VAR_TEMP
  iRetVal : INT ;	//return value as integer
  wRetVal : WORD ;	//return value as word
  Run : BOOL ;	//Unit in "RUN" mode
  EStopOK : BOOL ;	//Emergency Stop OK
  CIP : BOOL ;	//CIP Program Selected
  ComCIP : BOOL ;	//Communication with CIP Active
  xTmp : BOOL ;	//Temporary BOOL (free for general use)
  iTmp : INT ;	//Temporary INT (free for general use)
  rTmp : REAL ;	//Temporary REAL (free for general use)
  dTmp : DINT ;	//Temporary DINT (free for general use)
  UnitNo : INT ;	//Unit Number
  EquipmentID : INT ;	//Equipment ID
  Prid : DINT ;	//Process ID
  SFM36 : STRUCT 	// CIP Pump Mode
   I00 : BOOL ;	// Off
   I01 : BOOL ;	// Flow
   I02 : BOOL ;	// Pressure
   I03 : BOOL ;	// Fix Speed
   I04 : BOOL ;
   I05 : BOOL ;
   I06 : BOOL ;
   I07 : BOOL ;
   I08 : BOOL ;
   I09 : BOOL ;
   I10 : BOOL ;
   I11 : BOOL ;
   I12 : BOOL ;
   I13 : BOOL ;
   I14 : BOOL ;
   I15 : BOOL ;
   I16 : BOOL ;
   I17 : BOOL ;
   I18 : BOOL ;
   I19 : BOOL ;
   I20 : BOOL ;
   I21 : BOOL ;
   I22 : BOOL ;
   I23 : BOOL ;
   I24 : BOOL ;
   I25 : BOOL ;
   I26 : BOOL ;
   I27 : BOOL ;
   I28 : BOOL ;
   I29 : BOOL ;
   I30 : BOOL ;
   I31 : BOOL ;
  END_STRUCT ;
END_VAR
BEGIN
NETWORK
TITLE =general

      SET   ;

// unit & equipment number ---------------------------------------------------
      L     DB4210.DBW    0;
      T     #UnitNo;

      L     DB4215.DBW   14;
      L     1000;
      *I    ;
      L     #UnitNo;
      +I    ;
      T     #EquipmentID;

// CIP ----------------------------------------------------------------------
      L     DB4215.DBW   18;
      L     0;
      <I    ;
      =     #CIP;

// Communicating Units-------------------------------------------------------
      L     DB4215.DBD   10;
      L     DB4215.DBD  106;
      ==D   ;
      =     #ComCIP;

// emergency OK -------------------------------------------------------------
      A     DB4215.DBX   75.0; //General Emergency Stop OK
      CLR   ;
      =     #EStopOK;

NETWORK
TITLE =read other unit's data

      SET   ;

// ... General Unit ----------/

      CALL FC   563 (
           ActReq                   := M    101.0,
           PLCNo                    := 3,
           SourceUnitNo             := 99,
           IsTUnit                  := FALSE,
           DstComDRec               := DB4215.GEN,
           RET_VAL                  := #wRetVal);


NETWORK
TITLE =remote start

      SET   ;
// !!! insert correct condition of unit start !!!
      A     DB4211.DBX   15.0;
      A     DB4211.DBX   17.4;
      CLR   ;
      JCN   Strt;
      L     DB4215.DBD   10;
//L        L#-1;                            // Prid negative to start on its own
      T     #Prid;

      CALL FC    48 (
           UnitNo                   := #UnitNo,
           PrId                     := #Prid,
           Run                      := DB4211.DBX   17.4,
           PrIdTransfer             := TRUE,
           Start                    := TRUE,
           RetVal                   := #wRetVal);
Strt: NOP   0;
NETWORK
TITLE =external releases

      SET   ;

NETWORK
TITLE =write own unit data

      SET   ;

//-- CIP Communication ---------------------------------------
      AN    DB4211.DBX   15.0;
//      AN "U121SeqD".Seq.PO.B30 // CIP Active (Slave)
      A     #ComCIP;
      JCN   NCIP;
//Conductivity CIP Return
      L     DB4215.DBD  150;
      T     DB4211.DBD  626;

//Temperature CIP Return
      L     DB4215.DBD  146;
      T     DB4211.DBD  594;

//CIP Prerun Pump SP

      CALL FC    45 (
           SFM                      := DB4211.DBD  686,
           Indexes                  := #SFM36);


      L     0.000000e+000;
      A     #SFM36.I01;
      =     DB4215.DBX  171.7;
      JCN   pfc;
      L     DB4211.DBD  654;
pfc:  NOP   0;
      A     #SFM36.I02;
      =     DB4215.DBX  172.0;
      JCN   ppc;
      L     DB4211.DBD  670;
ppc:  NOP   0;
      A     #SFM36.I03;
      =     DB4215.DBX  171.6;
      JCN   pxc;
      L     DB4211.DBD  574;
pxc:  NOP   0;
      T     DB4215.DBD  182;

//CIP Return
      L     DB4211.DBD  558;
      T     DB4215.DBD  186;
      L     DB4215.DBD  138;
      T     DB4211.DBD  562;

//CIP Prerun
      L     DB4211.DBD  542;
      T     DB4215.DBD  190;
      L     DB4215.DBD  142;
      T     DB4211.DBD  546;

// Write Own Data to CIP
      L     DB4215.DBD   10;
      T     DB4215.DBD  154;

      L     DB4215.DBW   14;
      T     DB4215.DBW  158;

      L     DB4215.DBW   16;
      T     DB4215.DBW  160;

      L     DB4215.DBW   18;
      T     DB4215.DBW  162;

      L     DB4215.DBW   20;
      T     DB4215.DBW  164;

      L     DB4215.DBW   22;
      T     DB4215.DBW  166;

      A     DB4215.DBX   24.0;
      =     DB4215.DBX  168.0;

      A     DB4215.DBX   24.1;
      =     DB4215.DBX  168.1;

      A     DB4215.DBX   24.2;
      =     DB4215.DBX  168.2;

      A     DB4215.DBX   24.3;
      =     DB4215.DBX  168.3;

      A     DB4215.DBX   24.4;
      =     DB4215.DBX  168.4;

      A     DB4215.DBX   24.5;
      =     DB4215.DBX  168.5;

      A     DB4215.DBX   24.6;
      =     DB4215.DBX  168.6;

      A     DB4215.DBX   24.7;
      =     DB4215.DBX  168.7;

// Copy Data to CIP
      CALL SFC   20 (
           SRCBLK                   := DB4215.ToCIP,
           RET_VAL                  := #iRetVal,
           DSTBLK                   := DB4215.ToCIP);

NCIP: NOP   0;

//Empty Signal
//A     "U121SpID".SpI.Sig //!!!! Insert correct Empty Signal !!!
      CLR   ;
      =     DB4215.DBX   26.5;

//Full Signal
//A     "U121SpID".SpI.Sig //!!!! Insert correct Full Signal !!!
      CLR   ;
      =     DB4215.DBX   26.2;

//CIP Program Selected
      A     #CIP;
      =     DB4215.DBX   27.1;

// Emergency Stop
      A     #EStopOK; //If needed add or replace with own SpI
      =     DB4215.DBX   27.0; //Emergency Stop OK


NETWORK
TITLE = read from other unit data



END_FUNCTION_BLOCK

FUNCTION_BLOCK FB 4225
TITLE =U122: Planung Transfer VE2
FAMILY : BOTEC_F1
NAME : U122Comm
VERSION : 0.1


VAR_TEMP
  iRetVal : INT ;	//return value as integer
  wRetVal : WORD ;	//return value as word
  Run : BOOL ;	//Unit in "RUN" mode
  EStopOK : BOOL ;	//Emergency Stop OK
  CIP : BOOL ;	//CIP Program Selected
  ComCIP : BOOL ;	//Communication with CIP Active
  xTmp : BOOL ;	//Temporary BOOL (free for general use)
  iTmp : INT ;	//Temporary INT (free for general use)
  rTmp : REAL ;	//Temporary REAL (free for general use)
  dTmp : DINT ;	//Temporary DINT (free for general use)
  UnitNo : INT ;	//Unit Number
  EquipmentID : INT ;	//Equipment ID
  Prid : DINT ;	//Process ID
  SFM36 : STRUCT 	// CIP Pump Mode
   I00 : BOOL ;	// Off
   I01 : BOOL ;	// Flow
   I02 : BOOL ;	// Pressure
   I03 : BOOL ;	// Fix Speed
   I04 : BOOL ;
   I05 : BOOL ;
   I06 : BOOL ;
   I07 : BOOL ;
   I08 : BOOL ;
   I09 : BOOL ;
   I10 : BOOL ;
   I11 : BOOL ;
   I12 : BOOL ;
   I13 : BOOL ;
   I14 : BOOL ;
   I15 : BOOL ;
   I16 : BOOL ;
   I17 : BOOL ;
   I18 : BOOL ;
   I19 : BOOL ;
   I20 : BOOL ;
   I21 : BOOL ;
   I22 : BOOL ;
   I23 : BOOL ;
   I24 : BOOL ;
   I25 : BOOL ;
   I26 : BOOL ;
   I27 : BOOL ;
   I28 : BOOL ;
   I29 : BOOL ;
   I30 : BOOL ;
   I31 : BOOL ;
  END_STRUCT ;
END_VAR
BEGIN
NETWORK
TITLE =general

      SET   ;

// unit & equipment number ---------------------------------------------------
      L     DB4220.DBW    0;
      T     #UnitNo;

      L     DB4225.DBW   14;
      L     1000;
      *I    ;
      L     #UnitNo;
      +I    ;
      T     #EquipmentID;

// CIP ----------------------------------------------------------------------
      L     DB4225.DBW   18;
      L     0;
      <I    ;
      =     #CIP;

// Communicating Units-------------------------------------------------------
      L     DB4225.DBD   10;
      L     DB4225.DBD  106;
      ==D   ;
      =     #ComCIP;

// emergency OK -------------------------------------------------------------
      A     DB4225.DBX   75.0; //General Emergency Stop OK
      CLR   ;
      =     #EStopOK;

NETWORK
TITLE =read other unit's data

      SET   ;

// ... General Unit ----------/

      CALL FC   563 (
           ActReq                   := M    101.0,
           PLCNo                    := 3,
           SourceUnitNo             := 99,
           IsTUnit                  := FALSE,
           DstComDRec               := DB4225.GEN,
           RET_VAL                  := #wRetVal);

NETWORK
TITLE =remote start

      SET   ;
// !!! insert correct condition of unit start !!!
      A     DB4221.DBX   15.0;
      A     DB4221.DBX   17.4;
      CLR   ;
      JCN   Strt;
      L     DB4225.DBD   10;
//L        L#-1;                            // Prid negative to start on its own
      T     #Prid;

      CALL FC    48 (
           UnitNo                   := #UnitNo,
           PrId                     := #Prid,
           Run                      := DB4221.DBX   17.4,
           PrIdTransfer             := TRUE,
           Start                    := TRUE,
           RetVal                   := #wRetVal);
Strt: NOP   0;
NETWORK
TITLE =external releases

      SET   ;

NETWORK
TITLE =write own unit data

      SET   ;

//-- CIP Communication ---------------------------------------
      AN    DB4221.DBX   15.0;
//      AN "U122SeqD".Seq.PO.B30 // CIP Active (Slave)
      A     #ComCIP;
      JCN   NCIP;
//Conductivity CIP Return
      L     DB4225.DBD  150;
      T     DB4221.DBD  626;

//Temperature CIP Return
      L     DB4225.DBD  146;
      T     DB4221.DBD  594;

//CIP Prerun Pump SP

      CALL FC    45 (
           SFM                      := DB4221.DBD  686,
           Indexes                  := #SFM36);


      L     0.000000e+000;
      A     #SFM36.I01;
      =     DB4225.DBX  171.7;
      JCN   pfc;
      L     DB4221.DBD  654;
pfc:  NOP   0;
      A     #SFM36.I02;
      =     DB4225.DBX  172.0;
      JCN   ppc;
      L     DB4221.DBD  670;
ppc:  NOP   0;
      A     #SFM36.I03;
      =     DB4225.DBX  171.6;
      JCN   pxc;
      L     DB4221.DBD  574;
pxc:  NOP   0;
      T     DB4225.DBD  182;

//CIP Return
      L     DB4221.DBD  558;
      T     DB4225.DBD  186;
      L     DB4225.DBD  138;
      T     DB4221.DBD  562;

//CIP Prerun
      L     DB4221.DBD  542;
      T     DB4225.DBD  190;
      L     DB4225.DBD  142;
      T     DB4221.DBD  546;

// Write Own Data to CIP
      L     DB4225.DBD   10;
      T     DB4225.DBD  154;

      L     DB4225.DBW   14;
      T     DB4225.DBW  158;

      L     DB4225.DBW   16;
      T     DB4225.DBW  160;

      L     DB4225.DBW   18;
      T     DB4225.DBW  162;

      L     DB4225.DBW   20;
      T     DB4225.DBW  164;

      L     DB4225.DBW   22;
      T     DB4225.DBW  166;

      A     DB4225.DBX   24.0;
      =     DB4225.DBX  168.0;

      A     DB4225.DBX   24.1;
      =     DB4225.DBX  168.1;

      A     DB4225.DBX   24.2;
      =     DB4225.DBX  168.2;

      A     DB4225.DBX   24.3;
      =     DB4225.DBX  168.3;

      A     DB4225.DBX   24.4;
      =     DB4225.DBX  168.4;

      A     DB4225.DBX   24.5;
      =     DB4225.DBX  168.5;

      A     DB4225.DBX   24.6;
      =     DB4225.DBX  168.6;

      A     DB4225.DBX   24.7;
      =     DB4225.DBX  168.7;

// Copy Data to CIP
      CALL SFC   20 (
           SRCBLK                   := DB4225.ToCIP,
           RET_VAL                  := #iRetVal,
           DSTBLK                   := DB4225.ToCIP);

NCIP: NOP   0;

//Empty Signal
//A     "U122SpID".SpI.Sig //!!!! Insert correct Empty Signal !!!
      CLR   ;
      =     DB4225.DBX   26.5;

//Full Signal
//A     "U122SpID".SpI.Sig //!!!! Insert correct Full Signal !!!
      CLR   ;
      =     DB4225.DBX   26.2;

//CIP Program Selected
      A     #CIP;
      =     DB4225.DBX   27.1;

// Emergency Stop
      A     #EStopOK; //If needed add or replace with own SpI
      =     DB4225.DBX   27.0; //Emergency Stop OK


NETWORK
TITLE = read from other unit data



END_FUNCTION_BLOCK

FUNCTION_BLOCK FB 4255
TITLE =U125: Planung Transfer A
FAMILY : BOTEC_F1
NAME : U125Comm
VERSION : 0.1


VAR_TEMP
  iRetVal : INT ;	//return value as integer
  wRetVal : WORD ;	//return value as word
  Run : BOOL ;	//Unit in "RUN" mode
  EStopOK : BOOL ;	//Emergency Stop OK
  CIP : BOOL ;	//CIP Program Selected
  ComCIP : BOOL ;	//Communication with CIP Active
  xTmp : BOOL ;	//Temporary BOOL (free for general use)
  iTmp : INT ;	//Temporary INT (free for general use)
  rTmp : REAL ;	//Temporary REAL (free for general use)
  dTmp : DINT ;	//Temporary DINT (free for general use)
  UnitNo : INT ;	//Unit Number
  EquipmentID : INT ;	//Equipment ID
  Prid : DINT ;	//Process ID
  SFM36 : STRUCT 	// CIP Pump Mode
   I00 : BOOL ;	// Off
   I01 : BOOL ;	// Flow
   I02 : BOOL ;	// Pressure
   I03 : BOOL ;	// Fix Speed
   I04 : BOOL ;
   I05 : BOOL ;
   I06 : BOOL ;
   I07 : BOOL ;
   I08 : BOOL ;
   I09 : BOOL ;
   I10 : BOOL ;
   I11 : BOOL ;
   I12 : BOOL ;
   I13 : BOOL ;
   I14 : BOOL ;
   I15 : BOOL ;
   I16 : BOOL ;
   I17 : BOOL ;
   I18 : BOOL ;
   I19 : BOOL ;
   I20 : BOOL ;
   I21 : BOOL ;
   I22 : BOOL ;
   I23 : BOOL ;
   I24 : BOOL ;
   I25 : BOOL ;
   I26 : BOOL ;
   I27 : BOOL ;
   I28 : BOOL ;
   I29 : BOOL ;
   I30 : BOOL ;
   I31 : BOOL ;
  END_STRUCT ;
END_VAR
BEGIN
NETWORK
TITLE =general

      SET   ;

// unit & equipment number ---------------------------------------------------
      L     DB4250.DBW    0;
      T     #UnitNo;

      L     DB4255.DBW   14;
      L     1000;
      *I    ;
      L     #UnitNo;
      +I    ;
      T     #EquipmentID;

// CIP ----------------------------------------------------------------------
      L     DB4255.DBW   18;
      L     0;
      <I    ;
      =     #CIP;

// Communicating Units-------------------------------------------------------
      L     DB4255.DBD   10;
      L     DB4255.DBD  106;
      ==D   ;
      =     #ComCIP;

// emergency OK -------------------------------------------------------------
      A     DB4255.DBX   75.0; //General Emergency Stop OK
      CLR   ;
      =     #EStopOK;

NETWORK
TITLE =read other unit's data

      SET   ;

// ... General Unit ----------/

      CALL FC   563 (
           ActReq                   := M    101.0,
           PLCNo                    := 3,
           SourceUnitNo             := 99,
           IsTUnit                  := FALSE,
           DstComDRec               := DB4255.GEN,
           RET_VAL                  := #wRetVal);

NETWORK
TITLE =remote start

      SET   ;
// !!! insert correct condition of unit start !!!
      A     DB4251.DBX   15.0;
      A     DB4251.DBX   17.4;
      CLR   ;
      JCN   Strt;
      L     DB4255.DBD   10;
//L        L#-1;                            // Prid negative to start on its own
      T     #Prid;

      CALL FC    48 (
           UnitNo                   := #UnitNo,
           PrId                     := #Prid,
           Run                      := DB4251.DBX   17.4,
           PrIdTransfer             := TRUE,
           Start                    := TRUE,
           RetVal                   := #wRetVal);
Strt: NOP   0;
NETWORK
TITLE =external releases

      SET   ;

NETWORK
TITLE =write own unit data

      SET   ;

//-- CIP Communication ---------------------------------------
      AN    DB4251.DBX   15.0;
//      AN "U125SeqD".Seq.PO.B30 // CIP Active (Slave)
      A     #ComCIP;
      JCN   NCIP;
//Conductivity CIP Return
      L     DB4255.DBD  150;
      T     DB4251.DBD  626;

//Temperature CIP Return
      L     DB4255.DBD  146;
      T     DB4251.DBD  594;

//CIP Prerun Pump SP

      CALL FC    45 (
           SFM                      := DB4251.DBD  686,
           Indexes                  := #SFM36);


      L     0.000000e+000;
      A     #SFM36.I01;
      =     DB4255.DBX  171.7;
      JCN   pfc;
      L     DB4251.DBD  654;
pfc:  NOP   0;
      A     #SFM36.I02;
      =     DB4255.DBX  172.0;
      JCN   ppc;
      L     DB4251.DBD  670;
ppc:  NOP   0;
      A     #SFM36.I03;
      =     DB4255.DBX  171.6;
      JCN   pxc;
      L     DB4251.DBD  574;
pxc:  NOP   0;
      T     DB4255.DBD  182;

//CIP Return
      L     DB4251.DBD  558;
      T     DB4255.DBD  186;
      L     DB4255.DBD  138;
      T     DB4251.DBD  562;

//CIP Prerun
      L     DB4251.DBD  542;
      T     DB4255.DBD  190;
      L     DB4255.DBD  142;
      T     DB4251.DBD  546;

// Write Own Data to CIP
      L     DB4255.DBD   10;
      T     DB4255.DBD  154;

      L     DB4255.DBW   14;
      T     DB4255.DBW  158;

      L     DB4255.DBW   16;
      T     DB4255.DBW  160;

      L     DB4255.DBW   18;
      T     DB4255.DBW  162;

      L     DB4255.DBW   20;
      T     DB4255.DBW  164;

      L     DB4255.DBW   22;
      T     DB4255.DBW  166;

      A     DB4255.DBX   24.0;
      =     DB4255.DBX  168.0;

      A     DB4255.DBX   24.1;
      =     DB4255.DBX  168.1;

      A     DB4255.DBX   24.2;
      =     DB4255.DBX  168.2;

      A     DB4255.DBX   24.3;
      =     DB4255.DBX  168.3;

      A     DB4255.DBX   24.4;
      =     DB4255.DBX  168.4;

      A     DB4255.DBX   24.5;
      =     DB4255.DBX  168.5;

      A     DB4255.DBX   24.6;
      =     DB4255.DBX  168.6;

      A     DB4255.DBX   24.7;
      =     DB4255.DBX  168.7;

// Copy Data to CIP
      CALL SFC   20 (
           SRCBLK                   := DB4255.ToCIP,
           RET_VAL                  := #iRetVal,
           DSTBLK                   := DB4255.ToCIP);

NCIP: NOP   0;

//Empty Signal
//A     "U125SpID".SpI.Sig //!!!! Insert correct Empty Signal !!!
      CLR   ;
      =     DB4255.DBX   26.5;

//Full Signal
//A     "U125SpID".SpI.Sig //!!!! Insert correct Full Signal !!!
      CLR   ;
      =     DB4255.DBX   26.2;

//CIP Program Selected
      A     #CIP;
      =     DB4255.DBX   27.1;

// Emergency Stop
      A     #EStopOK; //If needed add or replace with own SpI
      =     DB4255.DBX   27.0; //Emergency Stop OK


NETWORK
TITLE = read from other unit data



END_FUNCTION_BLOCK

FUNCTION_BLOCK FB 4265
TITLE =U126: Planung Transfer B
FAMILY : BOTEC_F1
NAME : U126Comm
VERSION : 0.1


VAR_TEMP
  iRetVal : INT ;	//return value as integer
  wRetVal : WORD ;	//return value as word
  Run : BOOL ;	//Unit in "RUN" mode
  EStopOK : BOOL ;	//Emergency Stop OK
  CIP : BOOL ;	//CIP Program Selected
  ComCIP : BOOL ;	//Communication with CIP Active
  xTmp : BOOL ;	//Temporary BOOL (free for general use)
  iTmp : INT ;	//Temporary INT (free for general use)
  rTmp : REAL ;	//Temporary REAL (free for general use)
  dTmp : DINT ;	//Temporary DINT (free for general use)
  UnitNo : INT ;	//Unit Number
  EquipmentID : INT ;	//Equipment ID
  Prid : DINT ;	//Process ID
  SFM36 : STRUCT 	// CIP Pump Mode
   I00 : BOOL ;	// Off
   I01 : BOOL ;	// Flow
   I02 : BOOL ;	// Pressure
   I03 : BOOL ;	// Fix Speed
   I04 : BOOL ;
   I05 : BOOL ;
   I06 : BOOL ;
   I07 : BOOL ;
   I08 : BOOL ;
   I09 : BOOL ;
   I10 : BOOL ;
   I11 : BOOL ;
   I12 : BOOL ;
   I13 : BOOL ;
   I14 : BOOL ;
   I15 : BOOL ;
   I16 : BOOL ;
   I17 : BOOL ;
   I18 : BOOL ;
   I19 : BOOL ;
   I20 : BOOL ;
   I21 : BOOL ;
   I22 : BOOL ;
   I23 : BOOL ;
   I24 : BOOL ;
   I25 : BOOL ;
   I26 : BOOL ;
   I27 : BOOL ;
   I28 : BOOL ;
   I29 : BOOL ;
   I30 : BOOL ;
   I31 : BOOL ;
  END_STRUCT ;
END_VAR
BEGIN
NETWORK
TITLE =general

      SET   ;

// unit & equipment number ---------------------------------------------------
      L     DB4260.DBW    0;
      T     #UnitNo;

      L     DB4265.DBW   14;
      L     1000;
      *I    ;
      L     #UnitNo;
      +I    ;
      T     #EquipmentID;

// CIP ----------------------------------------------------------------------
      L     DB4265.DBW   18;
      L     0;
      <I    ;
      =     #CIP;

// Communicating Units-------------------------------------------------------
      L     DB4265.DBD   10;
      L     DB4265.DBD  106;
      ==D   ;
      =     #ComCIP;

// emergency OK -------------------------------------------------------------
      A     DB4265.DBX   75.0; //General Emergency Stop OK
      CLR   ;
      =     #EStopOK;

NETWORK
TITLE =read other unit's data

      SET   ;

// ... General Unit ----------/

      CALL FC   563 (
           ActReq                   := M    101.0,
           PLCNo                    := 3,
           SourceUnitNo             := 99,
           IsTUnit                  := FALSE,
           DstComDRec               := DB4265.GEN,
           RET_VAL                  := #wRetVal);


NETWORK
TITLE =remote start

      SET   ;
// !!! insert correct condition of unit start !!!
      A     DB4261.DBX   15.0;
      A     DB4261.DBX   17.4;
      CLR   ;
      JCN   Strt;
      L     DB4265.DBD   10;
//L        L#-1;                            // Prid negative to start on its own
      T     #Prid;

      CALL FC    48 (
           UnitNo                   := #UnitNo,
           PrId                     := #Prid,
           Run                      := DB4261.DBX   17.4,
           PrIdTransfer             := TRUE,
           Start                    := TRUE,
           RetVal                   := #wRetVal);
Strt: NOP   0;
NETWORK
TITLE =external releases

      SET   ;

NETWORK
TITLE =write own unit data

      SET   ;

//-- CIP Communication ---------------------------------------
      AN    DB4261.DBX   15.0;
//      AN "U126SeqD".Seq.PO.B30 // CIP Active (Slave)
      A     #ComCIP;
      JCN   NCIP;
//Conductivity CIP Return
      L     DB4265.DBD  150;
      T     DB4261.DBD  626;

//Temperature CIP Return
      L     DB4265.DBD  146;
      T     DB4261.DBD  594;

//CIP Prerun Pump SP

      CALL FC    45 (
           SFM                      := DB4261.DBD  686,
           Indexes                  := #SFM36);


      L     0.000000e+000;
      A     #SFM36.I01;
      =     DB4265.DBX  171.7;
      JCN   pfc;
      L     DB4261.DBD  654;
pfc:  NOP   0;
      A     #SFM36.I02;
      =     DB4265.DBX  172.0;
      JCN   ppc;
      L     DB4261.DBD  670;
ppc:  NOP   0;
      A     #SFM36.I03;
      =     DB4265.DBX  171.6;
      JCN   pxc;
      L     DB4261.DBD  574;
pxc:  NOP   0;
      T     DB4265.DBD  182;

//CIP Return
      L     DB4261.DBD  558;
      T     DB4265.DBD  186;
      L     DB4265.DBD  138;
      T     DB4261.DBD  562;

//CIP Prerun
      L     DB4261.DBD  542;
      T     DB4265.DBD  190;
      L     DB4265.DBD  142;
      T     DB4261.DBD  546;

// Write Own Data to CIP
      L     DB4265.DBD   10;
      T     DB4265.DBD  154;

      L     DB4265.DBW   14;
      T     DB4265.DBW  158;

      L     DB4265.DBW   16;
      T     DB4265.DBW  160;

      L     DB4265.DBW   18;
      T     DB4265.DBW  162;

      L     DB4265.DBW   20;
      T     DB4265.DBW  164;

      L     DB4265.DBW   22;
      T     DB4265.DBW  166;

      A     DB4265.DBX   24.0;
      =     DB4265.DBX  168.0;

      A     DB4265.DBX   24.1;
      =     DB4265.DBX  168.1;

      A     DB4265.DBX   24.2;
      =     DB4265.DBX  168.2;

      A     DB4265.DBX   24.3;
      =     DB4265.DBX  168.3;

      A     DB4265.DBX   24.4;
      =     DB4265.DBX  168.4;

      A     DB4265.DBX   24.5;
      =     DB4265.DBX  168.5;

      A     DB4265.DBX   24.6;
      =     DB4265.DBX  168.6;

      A     DB4265.DBX   24.7;
      =     DB4265.DBX  168.7;

// Copy Data to CIP
      CALL SFC   20 (
           SRCBLK                   := DB4265.ToCIP,
           RET_VAL                  := #iRetVal,
           DSTBLK                   := DB4265.ToCIP);

NCIP: NOP   0;

//Empty Signal
//A     "U126SpID".SpI.Sig //!!!! Insert correct Empty Signal !!!
      CLR   ;
      =     DB4265.DBX   26.5;

//Full Signal
//A     "U126SpID".SpI.Sig //!!!! Insert correct Full Signal !!!
      CLR   ;
      =     DB4265.DBX   26.2;

//CIP Program Selected
      A     #CIP;
      =     DB4265.DBX   27.1;

// Emergency Stop
      A     #EStopOK; //If needed add or replace with own SpI
      =     DB4265.DBX   27.0; //Emergency Stop OK


NETWORK
TITLE = read from other unit data



END_FUNCTION_BLOCK

FUNCTION_BLOCK FB 4275
TITLE =U127: Planung Transfer CF
FAMILY : BOTEC_F1
NAME : U127Comm
VERSION : 0.1


VAR_TEMP
  iRetVal : INT ;	//return value as integer
  wRetVal : WORD ;	//return value as word
  Run : BOOL ;	//Unit in "RUN" mode
  EStopOK : BOOL ;	//Emergency Stop OK
  CIP : BOOL ;	//CIP Program Selected
  ComCIP : BOOL ;	//Communication with CIP Active
  xTmp : BOOL ;	//Temporary BOOL (free for general use)
  iTmp : INT ;	//Temporary INT (free for general use)
  rTmp : REAL ;	//Temporary REAL (free for general use)
  dTmp : DINT ;	//Temporary DINT (free for general use)
  UnitNo : INT ;	//Unit Number
  EquipmentID : INT ;	//Equipment ID
  Prid : DINT ;	//Process ID
  SFM36 : STRUCT 	// CIP Pump Mode
   I00 : BOOL ;	// Off
   I01 : BOOL ;	// Flow
   I02 : BOOL ;	// Pressure
   I03 : BOOL ;	// Fix Speed
   I04 : BOOL ;
   I05 : BOOL ;
   I06 : BOOL ;
   I07 : BOOL ;
   I08 : BOOL ;
   I09 : BOOL ;
   I10 : BOOL ;
   I11 : BOOL ;
   I12 : BOOL ;
   I13 : BOOL ;
   I14 : BOOL ;
   I15 : BOOL ;
   I16 : BOOL ;
   I17 : BOOL ;
   I18 : BOOL ;
   I19 : BOOL ;
   I20 : BOOL ;
   I21 : BOOL ;
   I22 : BOOL ;
   I23 : BOOL ;
   I24 : BOOL ;
   I25 : BOOL ;
   I26 : BOOL ;
   I27 : BOOL ;
   I28 : BOOL ;
   I29 : BOOL ;
   I30 : BOOL ;
   I31 : BOOL ;
  END_STRUCT ;
END_VAR
BEGIN
NETWORK
TITLE =general

      SET   ;

// unit & equipment number ---------------------------------------------------
      L     DB4270.DBW    0;
      T     #UnitNo;

      L     DB4275.DBW   14;
      L     1000;
      *I    ;
      L     #UnitNo;
      +I    ;
      T     #EquipmentID;

// CIP ----------------------------------------------------------------------
      L     DB4275.DBW   18;
      L     0;
      <I    ;
      =     #CIP;

// Communicating Units-------------------------------------------------------
      L     DB4275.DBD   10;
      L     DB4275.DBD  106;
      ==D   ;
      =     #ComCIP;

// emergency OK -------------------------------------------------------------
      A     DB4275.DBX   75.0; //General Emergency Stop OK
      CLR   ;
      =     #EStopOK;

NETWORK
TITLE =read other unit's data

      SET   ;

// ... General Unit ----------/

      CALL FC   563 (
           ActReq                   := M    101.0,
           PLCNo                    := 3,
           SourceUnitNo             := 99,
           IsTUnit                  := FALSE,
           DstComDRec               := DB4275.GEN,
           RET_VAL                  := #wRetVal);

NETWORK
TITLE =remote start

      SET   ;
// !!! insert correct condition of unit start !!!
      A     DB4271.DBX   15.0;
      A     DB4271.DBX   17.4;
      CLR   ;
      JCN   Strt;
      L     DB4275.DBD   10;
//L        L#-1;                            // Prid negative to start on its own
      T     #Prid;

      CALL FC    48 (
           UnitNo                   := #UnitNo,
           PrId                     := #Prid,
           Run                      := DB4271.DBX   17.4,
           PrIdTransfer             := TRUE,
           Start                    := TRUE,
           RetVal                   := #wRetVal);
Strt: NOP   0;
NETWORK
TITLE =external releases

      SET   ;

NETWORK
TITLE =write own unit data

      SET   ;

//-- CIP Communication ---------------------------------------
      AN    DB4271.DBX   15.0;
//      AN "U127SeqD".Seq.PO.B30 // CIP Active (Slave)
      A     #ComCIP;
      JCN   NCIP;
//Conductivity CIP Return
      L     DB4275.DBD  150;
      T     DB4271.DBD  626;

//Temperature CIP Return
      L     DB4275.DBD  146;
      T     DB4271.DBD  594;

//CIP Prerun Pump SP

      CALL FC    45 (
           SFM                      := DB4271.DBD  686,
           Indexes                  := #SFM36);


      L     0.000000e+000;
      A     #SFM36.I01;
      =     DB4275.DBX  171.7;
      JCN   pfc;
      L     DB4271.DBD  654;
pfc:  NOP   0;
      A     #SFM36.I02;
      =     DB4275.DBX  172.0;
      JCN   ppc;
      L     DB4271.DBD  670;
ppc:  NOP   0;
      A     #SFM36.I03;
      =     DB4275.DBX  171.6;
      JCN   pxc;
      L     DB4271.DBD  574;
pxc:  NOP   0;
      T     DB4275.DBD  182;

//CIP Return
      L     DB4271.DBD  558;
      T     DB4275.DBD  186;
      L     DB4275.DBD  138;
      T     DB4271.DBD  562;

//CIP Prerun
      L     DB4271.DBD  542;
      T     DB4275.DBD  190;
      L     DB4275.DBD  142;
      T     DB4271.DBD  546;

// Write Own Data to CIP
      L     DB4275.DBD   10;
      T     DB4275.DBD  154;

      L     DB4275.DBW   14;
      T     DB4275.DBW  158;

      L     DB4275.DBW   16;
      T     DB4275.DBW  160;

      L     DB4275.DBW   18;
      T     DB4275.DBW  162;

      L     DB4275.DBW   20;
      T     DB4275.DBW  164;

      L     DB4275.DBW   22;
      T     DB4275.DBW  166;

      A     DB4275.DBX   24.0;
      =     DB4275.DBX  168.0;

      A     DB4275.DBX   24.1;
      =     DB4275.DBX  168.1;

      A     DB4275.DBX   24.2;
      =     DB4275.DBX  168.2;

      A     DB4275.DBX   24.3;
      =     DB4275.DBX  168.3;

      A     DB4275.DBX   24.4;
      =     DB4275.DBX  168.4;

      A     DB4275.DBX   24.5;
      =     DB4275.DBX  168.5;

      A     DB4275.DBX   24.6;
      =     DB4275.DBX  168.6;

      A     DB4275.DBX   24.7;
      =     DB4275.DBX  168.7;

// Copy Data to CIP
      CALL SFC   20 (
           SRCBLK                   := DB4275.ToCIP,
           RET_VAL                  := #iRetVal,
           DSTBLK                   := DB4275.ToCIP);

NCIP: NOP   0;

//Empty Signal
//A     "U127SpID".SpI.Sig //!!!! Insert correct Empty Signal !!!
      CLR   ;
      =     DB4275.DBX   26.5;

//Full Signal
//A     "U127SpID".SpI.Sig //!!!! Insert correct Full Signal !!!
      CLR   ;
      =     DB4275.DBX   26.2;

//CIP Program Selected
      A     #CIP;
      =     DB4275.DBX   27.1;

// Emergency Stop
      A     #EStopOK; //If needed add or replace with own SpI
      =     DB4275.DBX   27.0; //Emergency Stop OK


NETWORK
TITLE = read from other unit data



END_FUNCTION_BLOCK

FUNCTION_BLOCK FB 4285
TITLE =U128: Planung Transfer C.1
FAMILY : BOTEC_F1
NAME : U128Comm
VERSION : 0.1


VAR_TEMP
  iRetVal : INT ;	//return value as integer
  wRetVal : WORD ;	//return value as word
  Run : BOOL ;	//Unit in "RUN" mode
  EStopOK : BOOL ;	//Emergency Stop OK
  CIP : BOOL ;	//CIP Program Selected
  ComCIP : BOOL ;	//Communication with CIP Active
  xTmp : BOOL ;	//Temporary BOOL (free for general use)
  iTmp : INT ;	//Temporary INT (free for general use)
  rTmp : REAL ;	//Temporary REAL (free for general use)
  dTmp : DINT ;	//Temporary DINT (free for general use)
  UnitNo : INT ;	//Unit Number
  EquipmentID : INT ;	//Equipment ID
  Prid : DINT ;	//Process ID
  SFM36 : STRUCT 	// CIP Pump Mode
   I00 : BOOL ;	// Off
   I01 : BOOL ;	// Flow
   I02 : BOOL ;	// Pressure
   I03 : BOOL ;	// Fix Speed
   I04 : BOOL ;
   I05 : BOOL ;
   I06 : BOOL ;
   I07 : BOOL ;
   I08 : BOOL ;
   I09 : BOOL ;
   I10 : BOOL ;
   I11 : BOOL ;
   I12 : BOOL ;
   I13 : BOOL ;
   I14 : BOOL ;
   I15 : BOOL ;
   I16 : BOOL ;
   I17 : BOOL ;
   I18 : BOOL ;
   I19 : BOOL ;
   I20 : BOOL ;
   I21 : BOOL ;
   I22 : BOOL ;
   I23 : BOOL ;
   I24 : BOOL ;
   I25 : BOOL ;
   I26 : BOOL ;
   I27 : BOOL ;
   I28 : BOOL ;
   I29 : BOOL ;
   I30 : BOOL ;
   I31 : BOOL ;
  END_STRUCT ;
END_VAR
BEGIN
NETWORK
TITLE =general

      SET   ;

// unit & equipment number ---------------------------------------------------
      L     DB4280.DBW    0;
      T     #UnitNo;

      L     DB4285.DBW   14;
      L     1000;
      *I    ;
      L     #UnitNo;
      +I    ;
      T     #EquipmentID;

// CIP ----------------------------------------------------------------------
      L     DB4285.DBW   18;
      L     0;
      <I    ;
      =     #CIP;

// Communicating Units-------------------------------------------------------
      L     DB4285.DBD   10;
      L     DB4285.DBD  106;
      ==D   ;
      =     #ComCIP;

// emergency OK -------------------------------------------------------------
      A     DB4285.DBX   75.0; //General Emergency Stop OK
      CLR   ;
      =     #EStopOK;

NETWORK
TITLE =read other unit's data

      SET   ;

// ... General Unit ----------/

      CALL FC   563 (
           ActReq                   := M    101.0,
           PLCNo                    := 3,
           SourceUnitNo             := 99,
           IsTUnit                  := FALSE,
           DstComDRec               := DB4285.GEN,
           RET_VAL                  := #wRetVal);


NETWORK
TITLE =remote start

      SET   ;
// !!! insert correct condition of unit start !!!
      A     DB4281.DBX   15.0;
      A     DB4281.DBX   17.4;
      CLR   ;
      JCN   Strt;
      L     DB4285.DBD   10;
//L        L#-1;                            // Prid negative to start on its own
      T     #Prid;

      CALL FC    48 (
           UnitNo                   := #UnitNo,
           PrId                     := #Prid,
           Run                      := DB4281.DBX   17.4,
           PrIdTransfer             := TRUE,
           Start                    := TRUE,
           RetVal                   := #wRetVal);
Strt: NOP   0;
NETWORK
TITLE =external releases

      SET   ;

NETWORK
TITLE =write own unit data

      SET   ;

//-- CIP Communication ---------------------------------------
      AN    DB4281.DBX   15.0;
//      AN "U128SeqD".Seq.PO.B30 // CIP Active (Slave)
      A     #ComCIP;
      JCN   NCIP;
//Conductivity CIP Return
      L     DB4285.DBD  150;
      T     DB4281.DBD  626;

//Temperature CIP Return
      L     DB4285.DBD  146;
      T     DB4281.DBD  594;

//CIP Prerun Pump SP

      CALL FC    45 (
           SFM                      := DB4281.DBD  686,
           Indexes                  := #SFM36);


      L     0.000000e+000;
      A     #SFM36.I01;
      =     DB4285.DBX  171.7;
      JCN   pfc;
      L     DB4281.DBD  654;
pfc:  NOP   0;
      A     #SFM36.I02;
      =     DB4285.DBX  172.0;
      JCN   ppc;
      L     DB4281.DBD  670;
ppc:  NOP   0;
      A     #SFM36.I03;
      =     DB4285.DBX  171.6;
      JCN   pxc;
      L     DB4281.DBD  574;
pxc:  NOP   0;
      T     DB4285.DBD  182;

//CIP Return
      L     DB4281.DBD  558;
      T     DB4285.DBD  186;
      L     DB4285.DBD  138;
      T     DB4281.DBD  562;

//CIP Prerun
      L     DB4281.DBD  542;
      T     DB4285.DBD  190;
      L     DB4285.DBD  142;
      T     DB4281.DBD  546;

// Write Own Data to CIP
      L     DB4285.DBD   10;
      T     DB4285.DBD  154;

      L     DB4285.DBW   14;
      T     DB4285.DBW  158;

      L     DB4285.DBW   16;
      T     DB4285.DBW  160;

      L     DB4285.DBW   18;
      T     DB4285.DBW  162;

      L     DB4285.DBW   20;
      T     DB4285.DBW  164;

      L     DB4285.DBW   22;
      T     DB4285.DBW  166;

      A     DB4285.DBX   24.0;
      =     DB4285.DBX  168.0;

      A     DB4285.DBX   24.1;
      =     DB4285.DBX  168.1;

      A     DB4285.DBX   24.2;
      =     DB4285.DBX  168.2;

      A     DB4285.DBX   24.3;
      =     DB4285.DBX  168.3;

      A     DB4285.DBX   24.4;
      =     DB4285.DBX  168.4;

      A     DB4285.DBX   24.5;
      =     DB4285.DBX  168.5;

      A     DB4285.DBX   24.6;
      =     DB4285.DBX  168.6;

      A     DB4285.DBX   24.7;
      =     DB4285.DBX  168.7;

// Copy Data to CIP
      CALL SFC   20 (
           SRCBLK                   := DB4285.ToCIP,
           RET_VAL                  := #iRetVal,
           DSTBLK                   := DB4285.ToCIP);

NCIP: NOP   0;

//Empty Signal
//A     "U128SpID".SpI.Sig //!!!! Insert correct Empty Signal !!!
      CLR   ;
      =     DB4285.DBX   26.5;

//Full Signal
//A     "U128SpID".SpI.Sig //!!!! Insert correct Full Signal !!!
      CLR   ;
      =     DB4285.DBX   26.2;

//CIP Program Selected
      A     #CIP;
      =     DB4285.DBX   27.1;

// Emergency Stop
      A     #EStopOK; //If needed add or replace with own SpI
      =     DB4285.DBX   27.0; //Emergency Stop OK


NETWORK
TITLE = read from other unit data



END_FUNCTION_BLOCK

FUNCTION_BLOCK FB 4295
TITLE =U129: Planung Transfer B6F
FAMILY : BOTEC_F1
NAME : U129Comm
VERSION : 0.1


VAR_TEMP
  iRetVal : INT ;	//return value as integer
  wRetVal : WORD ;	//return value as word
  Run : BOOL ;	//Unit in "RUN" mode
  EStopOK : BOOL ;	//Emergency Stop OK
  CIP : BOOL ;	//CIP Program Selected
  ComCIP : BOOL ;	//Communication with CIP Active
  xTmp : BOOL ;	//Temporary BOOL (free for general use)
  iTmp : INT ;	//Temporary INT (free for general use)
  rTmp : REAL ;	//Temporary REAL (free for general use)
  dTmp : DINT ;	//Temporary DINT (free for general use)
  UnitNo : INT ;	//Unit Number
  EquipmentID : INT ;	//Equipment ID
  Prid : DINT ;	//Process ID
  SFM36 : STRUCT 	// CIP Pump Mode
   I00 : BOOL ;	// Off
   I01 : BOOL ;	// Flow
   I02 : BOOL ;	// Pressure
   I03 : BOOL ;	// Fix Speed
   I04 : BOOL ;
   I05 : BOOL ;
   I06 : BOOL ;
   I07 : BOOL ;
   I08 : BOOL ;
   I09 : BOOL ;
   I10 : BOOL ;
   I11 : BOOL ;
   I12 : BOOL ;
   I13 : BOOL ;
   I14 : BOOL ;
   I15 : BOOL ;
   I16 : BOOL ;
   I17 : BOOL ;
   I18 : BOOL ;
   I19 : BOOL ;
   I20 : BOOL ;
   I21 : BOOL ;
   I22 : BOOL ;
   I23 : BOOL ;
   I24 : BOOL ;
   I25 : BOOL ;
   I26 : BOOL ;
   I27 : BOOL ;
   I28 : BOOL ;
   I29 : BOOL ;
   I30 : BOOL ;
   I31 : BOOL ;
  END_STRUCT ;
END_VAR
BEGIN
NETWORK
TITLE =general

      SET   ;

// unit & equipment number ---------------------------------------------------
      L     DB4290.DBW    0;
      T     #UnitNo;

      L     DB4295.DBW   14;
      L     1000;
      *I    ;
      L     #UnitNo;
      +I    ;
      T     #EquipmentID;

// CIP ----------------------------------------------------------------------
      L     DB4295.DBW   18;
      L     0;
      <I    ;
      =     #CIP;

// Communicating Units-------------------------------------------------------
      L     DB4295.DBD   10;
      L     DB4295.DBD  106;
      ==D   ;
      =     #ComCIP;

// emergency OK -------------------------------------------------------------
      A     DB4295.DBX   75.0; //General Emergency Stop OK
      CLR   ;
      =     #EStopOK;

NETWORK
TITLE =read other unit's data

      SET   ;

// ... General Unit ----------/

      CALL FC   563 (
           ActReq                   := M    101.0,
           PLCNo                    := 3,
           SourceUnitNo             := 99,
           IsTUnit                  := FALSE,
           DstComDRec               := DB4295.GEN,
           RET_VAL                  := #wRetVal);


NETWORK
TITLE =remote start

      SET   ;
// !!! insert correct condition of unit start !!!
      A     DB4291.DBX   15.0;
      A     DB4291.DBX   17.4;
      CLR   ;
      JCN   Strt;
      L     DB4295.DBD   10;
//L        L#-1;                            // Prid negative to start on its own
      T     #Prid;

      CALL FC    48 (
           UnitNo                   := #UnitNo,
           PrId                     := #Prid,
           Run                      := DB4291.DBX   17.4,
           PrIdTransfer             := TRUE,
           Start                    := TRUE,
           RetVal                   := #wRetVal);
Strt: NOP   0;
NETWORK
TITLE =external releases

      SET   ;

NETWORK
TITLE =write own unit data

      SET   ;

//-- CIP Communication ---------------------------------------
      AN    DB4291.DBX   15.0;
//      AN "U129SeqD".Seq.PO.B30 // CIP Active (Slave)
      A     #ComCIP;
      JCN   NCIP;
//Conductivity CIP Return
      L     DB4295.DBD  150;
      T     DB4291.DBD  626;

//Temperature CIP Return
      L     DB4295.DBD  146;
      T     DB4291.DBD  594;

//CIP Prerun Pump SP

      CALL FC    45 (
           SFM                      := DB4291.DBD  686,
           Indexes                  := #SFM36);


      L     0.000000e+000;
      A     #SFM36.I01;
      =     DB4295.DBX  171.7;
      JCN   pfc;
      L     DB4291.DBD  654;
pfc:  NOP   0;
      A     #SFM36.I02;
      =     DB4295.DBX  172.0;
      JCN   ppc;
      L     DB4291.DBD  670;
ppc:  NOP   0;
      A     #SFM36.I03;
      =     DB4295.DBX  171.6;
      JCN   pxc;
      L     DB4291.DBD  574;
pxc:  NOP   0;
      T     DB4295.DBD  182;

//CIP Return
      L     DB4291.DBD  558;
      T     DB4295.DBD  186;
      L     DB4295.DBD  138;
      T     DB4291.DBD  562;

//CIP Prerun
      L     DB4291.DBD  542;
      T     DB4295.DBD  190;
      L     DB4295.DBD  142;
      T     DB4291.DBD  546;

// Write Own Data to CIP
      L     DB4295.DBD   10;
      T     DB4295.DBD  154;

      L     DB4295.DBW   14;
      T     DB4295.DBW  158;

      L     DB4295.DBW   16;
      T     DB4295.DBW  160;

      L     DB4295.DBW   18;
      T     DB4295.DBW  162;

      L     DB4295.DBW   20;
      T     DB4295.DBW  164;

      L     DB4295.DBW   22;
      T     DB4295.DBW  166;

      A     DB4295.DBX   24.0;
      =     DB4295.DBX  168.0;

      A     DB4295.DBX   24.1;
      =     DB4295.DBX  168.1;

      A     DB4295.DBX   24.2;
      =     DB4295.DBX  168.2;

      A     DB4295.DBX   24.3;
      =     DB4295.DBX  168.3;

      A     DB4295.DBX   24.4;
      =     DB4295.DBX  168.4;

      A     DB4295.DBX   24.5;
      =     DB4295.DBX  168.5;

      A     DB4295.DBX   24.6;
      =     DB4295.DBX  168.6;

      A     DB4295.DBX   24.7;
      =     DB4295.DBX  168.7;

// Copy Data to CIP
      CALL SFC   20 (
           SRCBLK                   := DB4295.ToCIP,
           RET_VAL                  := #iRetVal,
           DSTBLK                   := DB4295.ToCIP);

NCIP: NOP   0;

//Empty Signal
//A     "U129SpID".SpI.Sig //!!!! Insert correct Empty Signal !!!
      CLR   ;
      =     DB4295.DBX   26.5;

//Full Signal
//A     "U129SpID".SpI.Sig //!!!! Insert correct Full Signal !!!
      CLR   ;
      =     DB4295.DBX   26.2;

//CIP Program Selected
      A     #CIP;
      =     DB4295.DBX   27.1;

// Emergency Stop
      A     #EStopOK; //If needed add or replace with own SpI
      =     DB4295.DBX   27.0; //Emergency Stop OK


NETWORK
TITLE = read from other unit data



END_FUNCTION_BLOCK

FUNCTION_BLOCK FB 4305
TITLE =U130: Planung Transfer H6F
FAMILY : BOTEC_F1
NAME : U130Comm
VERSION : 0.1


VAR_TEMP
  iRetVal : INT ;	//return value as integer
  wRetVal : WORD ;	//return value as word
  Run : BOOL ;	//Unit in "RUN" mode
  EStopOK : BOOL ;	//Emergency Stop OK
  CIP : BOOL ;	//CIP Program Selected
  ComCIP : BOOL ;	//Communication with CIP Active
  xTmp : BOOL ;	//Temporary BOOL (free for general use)
  iTmp : INT ;	//Temporary INT (free for general use)
  rTmp : REAL ;	//Temporary REAL (free for general use)
  dTmp : DINT ;	//Temporary DINT (free for general use)
  UnitNo : INT ;	//Unit Number
  EquipmentID : INT ;	//Equipment ID
  Prid : DINT ;	//Process ID
  SFM36 : STRUCT 	// CIP Pump Mode
   I00 : BOOL ;	// Off
   I01 : BOOL ;	// Flow
   I02 : BOOL ;	// Pressure
   I03 : BOOL ;	// Fix Speed
   I04 : BOOL ;
   I05 : BOOL ;
   I06 : BOOL ;
   I07 : BOOL ;
   I08 : BOOL ;
   I09 : BOOL ;
   I10 : BOOL ;
   I11 : BOOL ;
   I12 : BOOL ;
   I13 : BOOL ;
   I14 : BOOL ;
   I15 : BOOL ;
   I16 : BOOL ;
   I17 : BOOL ;
   I18 : BOOL ;
   I19 : BOOL ;
   I20 : BOOL ;
   I21 : BOOL ;
   I22 : BOOL ;
   I23 : BOOL ;
   I24 : BOOL ;
   I25 : BOOL ;
   I26 : BOOL ;
   I27 : BOOL ;
   I28 : BOOL ;
   I29 : BOOL ;
   I30 : BOOL ;
   I31 : BOOL ;
  END_STRUCT ;
END_VAR
BEGIN
NETWORK
TITLE =general

      SET   ;

// unit & equipment number ---------------------------------------------------
      L     DB4300.DBW    0;
      T     #UnitNo;

      L     DB4305.DBW   14;
      L     1000;
      *I    ;
      L     #UnitNo;
      +I    ;
      T     #EquipmentID;

// CIP ----------------------------------------------------------------------
      L     DB4305.DBW   18;
      L     0;
      <I    ;
      =     #CIP;

// Communicating Units-------------------------------------------------------
      L     DB4305.DBD   10;
      L     DB4305.DBD  106;
      ==D   ;
      =     #ComCIP;

// emergency OK -------------------------------------------------------------
      A     DB4305.DBX   75.0; //General Emergency Stop OK
      CLR   ;
      =     #EStopOK;

NETWORK
TITLE =read other unit's data

      SET   ;

// ... General Unit ----------/

      CALL FC   563 (
           ActReq                   := M    101.0,
           PLCNo                    := 3,
           SourceUnitNo             := 99,
           IsTUnit                  := FALSE,
           DstComDRec               := DB4305.GEN,
           RET_VAL                  := #wRetVal);

NETWORK
TITLE =remote start

      SET   ;
// !!! insert correct condition of unit start !!!
      A     DB4301.DBX   15.0;
      A     DB4301.DBX   17.4;
      CLR   ;
      JCN   Strt;
      L     DB4305.DBD   10;
//L        L#-1;                            // Prid negative to start on its own
      T     #Prid;

      CALL FC    48 (
           UnitNo                   := #UnitNo,
           PrId                     := #Prid,
           Run                      := DB4301.DBX   17.4,
           PrIdTransfer             := TRUE,
           Start                    := TRUE,
           RetVal                   := #wRetVal);
Strt: NOP   0;
NETWORK
TITLE =external releases

      SET   ;

NETWORK
TITLE =write own unit data

      SET   ;

//-- CIP Communication ---------------------------------------
      AN    DB4301.DBX   15.0;
//      AN "U130SeqD".Seq.PO.B30 // CIP Active (Slave)
      A     #ComCIP;
      JCN   NCIP;
//Conductivity CIP Return
      L     DB4305.DBD  150;
      T     DB4301.DBD  626;

//Temperature CIP Return
      L     DB4305.DBD  146;
      T     DB4301.DBD  594;

//CIP Prerun Pump SP

      CALL FC    45 (
           SFM                      := DB4301.DBD  686,
           Indexes                  := #SFM36);


      L     0.000000e+000;
      A     #SFM36.I01;
      =     DB4305.DBX  171.7;
      JCN   pfc;
      L     DB4301.DBD  654;
pfc:  NOP   0;
      A     #SFM36.I02;
      =     DB4305.DBX  172.0;
      JCN   ppc;
      L     DB4301.DBD  670;
ppc:  NOP   0;
      A     #SFM36.I03;
      =     DB4305.DBX  171.6;
      JCN   pxc;
      L     DB4301.DBD  574;
pxc:  NOP   0;
      T     DB4305.DBD  182;

//CIP Return
      L     DB4301.DBD  558;
      T     DB4305.DBD  186;
      L     DB4305.DBD  138;
      T     DB4301.DBD  562;

//CIP Prerun
      L     DB4301.DBD  542;
      T     DB4305.DBD  190;
      L     DB4305.DBD  142;
      T     DB4301.DBD  546;

// Write Own Data to CIP
      L     DB4305.DBD   10;
      T     DB4305.DBD  154;

      L     DB4305.DBW   14;
      T     DB4305.DBW  158;

      L     DB4305.DBW   16;
      T     DB4305.DBW  160;

      L     DB4305.DBW   18;
      T     DB4305.DBW  162;

      L     DB4305.DBW   20;
      T     DB4305.DBW  164;

      L     DB4305.DBW   22;
      T     DB4305.DBW  166;

      A     DB4305.DBX   24.0;
      =     DB4305.DBX  168.0;

      A     DB4305.DBX   24.1;
      =     DB4305.DBX  168.1;

      A     DB4305.DBX   24.2;
      =     DB4305.DBX  168.2;

      A     DB4305.DBX   24.3;
      =     DB4305.DBX  168.3;

      A     DB4305.DBX   24.4;
      =     DB4305.DBX  168.4;

      A     DB4305.DBX   24.5;
      =     DB4305.DBX  168.5;

      A     DB4305.DBX   24.6;
      =     DB4305.DBX  168.6;

      A     DB4305.DBX   24.7;
      =     DB4305.DBX  168.7;

// Copy Data to CIP
      CALL SFC   20 (
           SRCBLK                   := DB4305.ToCIP,
           RET_VAL                  := #iRetVal,
           DSTBLK                   := DB4305.ToCIP);

NCIP: NOP   0;

//Empty Signal
//A     "U130SpID".SpI.Sig //!!!! Insert correct Empty Signal !!!
      CLR   ;
      =     DB4305.DBX   26.5;

//Full Signal
//A     "U130SpID".SpI.Sig //!!!! Insert correct Full Signal !!!
      CLR   ;
      =     DB4305.DBX   26.2;

//CIP Program Selected
      A     #CIP;
      =     DB4305.DBX   27.1;

// Emergency Stop
      A     #EStopOK; //If needed add or replace with own SpI
      =     DB4305.DBX   27.0; //Emergency Stop OK


NETWORK
TITLE = read from other unit data



END_FUNCTION_BLOCK

FUNCTION_BLOCK FB 4315
TITLE =U131: Planung Transfer J6F
FAMILY : BOTEC_F1
NAME : U131Comm
VERSION : 0.1


VAR_TEMP
  iRetVal : INT ;	//return value as integer
  wRetVal : WORD ;	//return value as word
  Run : BOOL ;	//Unit in "RUN" mode
  EStopOK : BOOL ;	//Emergency Stop OK
  CIP : BOOL ;	//CIP Program Selected
  ComCIP : BOOL ;	//Communication with CIP Active
  xTmp : BOOL ;	//Temporary BOOL (free for general use)
  iTmp : INT ;	//Temporary INT (free for general use)
  rTmp : REAL ;	//Temporary REAL (free for general use)
  dTmp : DINT ;	//Temporary DINT (free for general use)
  UnitNo : INT ;	//Unit Number
  EquipmentID : INT ;	//Equipment ID
  Prid : DINT ;	//Process ID
  SFM36 : STRUCT 	// CIP Pump Mode
   I00 : BOOL ;	// Off
   I01 : BOOL ;	// Flow
   I02 : BOOL ;	// Pressure
   I03 : BOOL ;	// Fix Speed
   I04 : BOOL ;
   I05 : BOOL ;
   I06 : BOOL ;
   I07 : BOOL ;
   I08 : BOOL ;
   I09 : BOOL ;
   I10 : BOOL ;
   I11 : BOOL ;
   I12 : BOOL ;
   I13 : BOOL ;
   I14 : BOOL ;
   I15 : BOOL ;
   I16 : BOOL ;
   I17 : BOOL ;
   I18 : BOOL ;
   I19 : BOOL ;
   I20 : BOOL ;
   I21 : BOOL ;
   I22 : BOOL ;
   I23 : BOOL ;
   I24 : BOOL ;
   I25 : BOOL ;
   I26 : BOOL ;
   I27 : BOOL ;
   I28 : BOOL ;
   I29 : BOOL ;
   I30 : BOOL ;
   I31 : BOOL ;
  END_STRUCT ;
END_VAR
BEGIN
NETWORK
TITLE =general

      SET   ;

// unit & equipment number ---------------------------------------------------
      L     DB4310.DBW    0;
      T     #UnitNo;

      L     DB4315.DBW   14;
      L     1000;
      *I    ;
      L     #UnitNo;
      +I    ;
      T     #EquipmentID;

// CIP ----------------------------------------------------------------------
      L     DB4315.DBW   18;
      L     0;
      <I    ;
      =     #CIP;

// Communicating Units-------------------------------------------------------
      L     DB4315.DBD   10;
      L     DB4315.DBD  106;
      ==D   ;
      =     #ComCIP;

// emergency OK -------------------------------------------------------------
      A     DB4315.DBX   75.0; //General Emergency Stop OK
      CLR   ;
      =     #EStopOK;

NETWORK
TITLE =read other unit's data

      SET   ;

// ... General Unit ----------/

      CALL FC   563 (
           ActReq                   := M    101.0,
           PLCNo                    := 3,
           SourceUnitNo             := 99,
           IsTUnit                  := FALSE,
           DstComDRec               := DB4315.GEN,
           RET_VAL                  := #wRetVal);


NETWORK
TITLE =remote start

      SET   ;
// !!! insert correct condition of unit start !!!
      A     DB4311.DBX   15.0;
      A     DB4311.DBX   17.4;
      CLR   ;
      JCN   Strt;
      L     DB4315.DBD   10;
//L        L#-1;                            // Prid negative to start on its own
      T     #Prid;

      CALL FC    48 (
           UnitNo                   := #UnitNo,
           PrId                     := #Prid,
           Run                      := DB4311.DBX   17.4,
           PrIdTransfer             := TRUE,
           Start                    := TRUE,
           RetVal                   := #wRetVal);
Strt: NOP   0;
NETWORK
TITLE =external releases

      SET   ;

NETWORK
TITLE =write own unit data

      SET   ;

//-- CIP Communication ---------------------------------------
      AN    DB4311.DBX   15.0;
//      AN "U131SeqD".Seq.PO.B30 // CIP Active (Slave)
      A     #ComCIP;
      JCN   NCIP;
//Conductivity CIP Return
      L     DB4315.DBD  150;
      T     DB4311.DBD  626;

//Temperature CIP Return
      L     DB4315.DBD  146;
      T     DB4311.DBD  594;

//CIP Prerun Pump SP

      CALL FC    45 (
           SFM                      := DB4311.DBD  686,
           Indexes                  := #SFM36);


      L     0.000000e+000;
      A     #SFM36.I01;
      =     DB4315.DBX  171.7;
      JCN   pfc;
      L     DB4311.DBD  654;
pfc:  NOP   0;
      A     #SFM36.I02;
      =     DB4315.DBX  172.0;
      JCN   ppc;
      L     DB4311.DBD  670;
ppc:  NOP   0;
      A     #SFM36.I03;
      =     DB4315.DBX  171.6;
      JCN   pxc;
      L     DB4311.DBD  574;
pxc:  NOP   0;
      T     DB4315.DBD  182;

//CIP Return
      L     DB4311.DBD  558;
      T     DB4315.DBD  186;
      L     DB4315.DBD  138;
      T     DB4311.DBD  562;

//CIP Prerun
      L     DB4311.DBD  542;
      T     DB4315.DBD  190;
      L     DB4315.DBD  142;
      T     DB4311.DBD  546;

// Write Own Data to CIP
      L     DB4315.DBD   10;
      T     DB4315.DBD  154;

      L     DB4315.DBW   14;
      T     DB4315.DBW  158;

      L     DB4315.DBW   16;
      T     DB4315.DBW  160;

      L     DB4315.DBW   18;
      T     DB4315.DBW  162;

      L     DB4315.DBW   20;
      T     DB4315.DBW  164;

      L     DB4315.DBW   22;
      T     DB4315.DBW  166;

      A     DB4315.DBX   24.0;
      =     DB4315.DBX  168.0;

      A     DB4315.DBX   24.1;
      =     DB4315.DBX  168.1;

      A     DB4315.DBX   24.2;
      =     DB4315.DBX  168.2;

      A     DB4315.DBX   24.3;
      =     DB4315.DBX  168.3;

      A     DB4315.DBX   24.4;
      =     DB4315.DBX  168.4;

      A     DB4315.DBX   24.5;
      =     DB4315.DBX  168.5;

      A     DB4315.DBX   24.6;
      =     DB4315.DBX  168.6;

      A     DB4315.DBX   24.7;
      =     DB4315.DBX  168.7;

// Copy Data to CIP
      CALL SFC   20 (
           SRCBLK                   := DB4315.ToCIP,
           RET_VAL                  := #iRetVal,
           DSTBLK                   := DB4315.ToCIP);

NCIP: NOP   0;

//Empty Signal
//A     "U131SpID".SpI.Sig //!!!! Insert correct Empty Signal !!!
      CLR   ;
      =     DB4315.DBX   26.5;

//Full Signal
//A     "U131SpID".SpI.Sig //!!!! Insert correct Full Signal !!!
      CLR   ;
      =     DB4315.DBX   26.2;

//CIP Program Selected
      A     #CIP;
      =     DB4315.DBX   27.1;

// Emergency Stop
      A     #EStopOK; //If needed add or replace with own SpI
      =     DB4315.DBX   27.0; //Emergency Stop OK


NETWORK
TITLE = read from other unit data



END_FUNCTION_BLOCK

FUNCTION_BLOCK FB 4325
TITLE =U132: Planung Transfer L6F
FAMILY : BOTEC_F1
NAME : U132Comm
VERSION : 0.1


VAR_TEMP
  iRetVal : INT ;	//return value as integer
  wRetVal : WORD ;	//return value as word
  Run : BOOL ;	//Unit in "RUN" mode
  EStopOK : BOOL ;	//Emergency Stop OK
  CIP : BOOL ;	//CIP Program Selected
  ComCIP : BOOL ;	//Communication with CIP Active
  xTmp : BOOL ;	//Temporary BOOL (free for general use)
  iTmp : INT ;	//Temporary INT (free for general use)
  rTmp : REAL ;	//Temporary REAL (free for general use)
  dTmp : DINT ;	//Temporary DINT (free for general use)
  UnitNo : INT ;	//Unit Number
  EquipmentID : INT ;	//Equipment ID
  Prid : DINT ;	//Process ID
  SFM36 : STRUCT 	// CIP Pump Mode
   I00 : BOOL ;	// Off
   I01 : BOOL ;	// Flow
   I02 : BOOL ;	// Pressure
   I03 : BOOL ;	// Fix Speed
   I04 : BOOL ;
   I05 : BOOL ;
   I06 : BOOL ;
   I07 : BOOL ;
   I08 : BOOL ;
   I09 : BOOL ;
   I10 : BOOL ;
   I11 : BOOL ;
   I12 : BOOL ;
   I13 : BOOL ;
   I14 : BOOL ;
   I15 : BOOL ;
   I16 : BOOL ;
   I17 : BOOL ;
   I18 : BOOL ;
   I19 : BOOL ;
   I20 : BOOL ;
   I21 : BOOL ;
   I22 : BOOL ;
   I23 : BOOL ;
   I24 : BOOL ;
   I25 : BOOL ;
   I26 : BOOL ;
   I27 : BOOL ;
   I28 : BOOL ;
   I29 : BOOL ;
   I30 : BOOL ;
   I31 : BOOL ;
  END_STRUCT ;
END_VAR
BEGIN
NETWORK
TITLE =general

      SET   ;

// unit & equipment number ---------------------------------------------------
      L     DB4320.DBW    0;
      T     #UnitNo;

      L     DB4325.DBW   14;
      L     1000;
      *I    ;
      L     #UnitNo;
      +I    ;
      T     #EquipmentID;

// CIP ----------------------------------------------------------------------
      L     DB4325.DBW   18;
      L     0;
      <I    ;
      =     #CIP;

// Communicating Units-------------------------------------------------------
      L     DB4325.DBD   10;
      L     DB4325.DBD  106;
      ==D   ;
      =     #ComCIP;

// emergency OK -------------------------------------------------------------
      A     DB4325.DBX   75.0; //General Emergency Stop OK
      CLR   ;
      =     #EStopOK;

NETWORK
TITLE =read other unit's data

      SET   ;

// ... General Unit ----------/

      CALL FC   563 (
           ActReq                   := M    101.0,
           PLCNo                    := 3,
           SourceUnitNo             := 99,
           IsTUnit                  := FALSE,
           DstComDRec               := DB4325.GEN,
           RET_VAL                  := #wRetVal);

NETWORK
TITLE =remote start

      SET   ;
// !!! insert correct condition of unit start !!!
      A     DB4321.DBX   15.0;
      A     DB4321.DBX   17.4;
      CLR   ;
      JCN   Strt;
      L     DB4325.DBD   10;
//L        L#-1;                            // Prid negative to start on its own
      T     #Prid;

      CALL FC    48 (
           UnitNo                   := #UnitNo,
           PrId                     := #Prid,
           Run                      := DB4321.DBX   17.4,
           PrIdTransfer             := TRUE,
           Start                    := TRUE,
           RetVal                   := #wRetVal);
Strt: NOP   0;
NETWORK
TITLE =external releases

      SET   ;

NETWORK
TITLE =write own unit data

      SET   ;

//-- CIP Communication ---------------------------------------
      AN    DB4321.DBX   15.0;
//      AN "U132SeqD".Seq.PO.B30 // CIP Active (Slave)
      A     #ComCIP;
      JCN   NCIP;
//Conductivity CIP Return
      L     DB4325.DBD  150;
      T     DB4321.DBD  626;

//Temperature CIP Return
      L     DB4325.DBD  146;
      T     DB4321.DBD  594;

//CIP Prerun Pump SP

      CALL FC    45 (
           SFM                      := DB4321.DBD  686,
           Indexes                  := #SFM36);


      L     0.000000e+000;
      A     #SFM36.I01;
      =     DB4325.DBX  171.7;
      JCN   pfc;
      L     DB4321.DBD  654;
pfc:  NOP   0;
      A     #SFM36.I02;
      =     DB4325.DBX  172.0;
      JCN   ppc;
      L     DB4321.DBD  670;
ppc:  NOP   0;
      A     #SFM36.I03;
      =     DB4325.DBX  171.6;
      JCN   pxc;
      L     DB4321.DBD  574;
pxc:  NOP   0;
      T     DB4325.DBD  182;

//CIP Return
      L     DB4321.DBD  558;
      T     DB4325.DBD  186;
      L     DB4325.DBD  138;
      T     DB4321.DBD  562;

//CIP Prerun
      L     DB4321.DBD  542;
      T     DB4325.DBD  190;
      L     DB4325.DBD  142;
      T     DB4321.DBD  546;

// Write Own Data to CIP
      L     DB4325.DBD   10;
      T     DB4325.DBD  154;

      L     DB4325.DBW   14;
      T     DB4325.DBW  158;

      L     DB4325.DBW   16;
      T     DB4325.DBW  160;

      L     DB4325.DBW   18;
      T     DB4325.DBW  162;

      L     DB4325.DBW   20;
      T     DB4325.DBW  164;

      L     DB4325.DBW   22;
      T     DB4325.DBW  166;

      A     DB4325.DBX   24.0;
      =     DB4325.DBX  168.0;

      A     DB4325.DBX   24.1;
      =     DB4325.DBX  168.1;

      A     DB4325.DBX   24.2;
      =     DB4325.DBX  168.2;

      A     DB4325.DBX   24.3;
      =     DB4325.DBX  168.3;

      A     DB4325.DBX   24.4;
      =     DB4325.DBX  168.4;

      A     DB4325.DBX   24.5;
      =     DB4325.DBX  168.5;

      A     DB4325.DBX   24.6;
      =     DB4325.DBX  168.6;

      A     DB4325.DBX   24.7;
      =     DB4325.DBX  168.7;

// Copy Data to CIP
      CALL SFC   20 (
           SRCBLK                   := DB4325.ToCIP,
           RET_VAL                  := #iRetVal,
           DSTBLK                   := DB4325.ToCIP);

NCIP: NOP   0;

//Empty Signal
//A     "U132SpID".SpI.Sig //!!!! Insert correct Empty Signal !!!
      CLR   ;
      =     DB4325.DBX   26.5;

//Full Signal
//A     "U132SpID".SpI.Sig //!!!! Insert correct Full Signal !!!
      CLR   ;
      =     DB4325.DBX   26.2;

//CIP Program Selected
      A     #CIP;
      =     DB4325.DBX   27.1;

// Emergency Stop
      A     #EStopOK; //If needed add or replace with own SpI
      =     DB4325.DBX   27.0; //Emergency Stop OK


NETWORK
TITLE = read from other unit data



END_FUNCTION_BLOCK

FUNCTION_BLOCK FB 4335
TITLE =U133: Planung Transfer B6
FAMILY : BOTEC_F1
NAME : U133Comm
VERSION : 0.1


VAR_TEMP
  iRetVal : INT ;	//return value as integer
  wRetVal : WORD ;	//return value as word
  Run : BOOL ;	//Unit in "RUN" mode
  EStopOK : BOOL ;	//Emergency Stop OK
  CIP : BOOL ;	//CIP Program Selected
  ComCIP : BOOL ;	//Communication with CIP Active
  xTmp : BOOL ;	//Temporary BOOL (free for general use)
  iTmp : INT ;	//Temporary INT (free for general use)
  rTmp : REAL ;	//Temporary REAL (free for general use)
  dTmp : DINT ;	//Temporary DINT (free for general use)
  UnitNo : INT ;	//Unit Number
  EquipmentID : INT ;	//Equipment ID
  Prid : DINT ;	//Process ID
  SFM36 : STRUCT 	// CIP Pump Mode
   I00 : BOOL ;	// Off
   I01 : BOOL ;	// Flow
   I02 : BOOL ;	// Pressure
   I03 : BOOL ;	// Fix Speed
   I04 : BOOL ;
   I05 : BOOL ;
   I06 : BOOL ;
   I07 : BOOL ;
   I08 : BOOL ;
   I09 : BOOL ;
   I10 : BOOL ;
   I11 : BOOL ;
   I12 : BOOL ;
   I13 : BOOL ;
   I14 : BOOL ;
   I15 : BOOL ;
   I16 : BOOL ;
   I17 : BOOL ;
   I18 : BOOL ;
   I19 : BOOL ;
   I20 : BOOL ;
   I21 : BOOL ;
   I22 : BOOL ;
   I23 : BOOL ;
   I24 : BOOL ;
   I25 : BOOL ;
   I26 : BOOL ;
   I27 : BOOL ;
   I28 : BOOL ;
   I29 : BOOL ;
   I30 : BOOL ;
   I31 : BOOL ;
  END_STRUCT ;
END_VAR
BEGIN
NETWORK
TITLE =general

      SET   ;

// unit & equipment number ---------------------------------------------------
      L     DB4330.DBW    0;
      T     #UnitNo;

      L     DB4335.DBW   14;
      L     1000;
      *I    ;
      L     #UnitNo;
      +I    ;
      T     #EquipmentID;

// CIP ----------------------------------------------------------------------
      L     DB4335.DBW   18;
      L     0;
      <I    ;
      =     #CIP;

// Communicating Units-------------------------------------------------------
      L     DB4335.DBD   10;
      L     DB4335.DBD  106;
      ==D   ;
      =     #ComCIP;

// emergency OK -------------------------------------------------------------
      A     DB4335.DBX   75.0; //General Emergency Stop OK
      CLR   ;
      =     #EStopOK;

NETWORK
TITLE =read other unit's data

      SET   ;

// ... General Unit ----------/

      CALL FC   563 (
           ActReq                   := M    101.0,
           PLCNo                    := 3,
           SourceUnitNo             := 99,
           IsTUnit                  := FALSE,
           DstComDRec               := DB4335.GEN,
           RET_VAL                  := #wRetVal);


NETWORK
TITLE =remote start

      SET   ;
// !!! insert correct condition of unit start !!!
      A     DB4331.DBX   15.0;
      A     DB4331.DBX   17.4;
      CLR   ;
      JCN   Strt;
      L     DB4335.DBD   10;
//L        L#-1;                            // Prid negative to start on its own
      T     #Prid;

      CALL FC    48 (
           UnitNo                   := #UnitNo,
           PrId                     := #Prid,
           Run                      := DB4331.DBX   17.4,
           PrIdTransfer             := TRUE,
           Start                    := TRUE,
           RetVal                   := #wRetVal);
Strt: NOP   0;
NETWORK
TITLE =external releases

      SET   ;

NETWORK
TITLE =write own unit data

      SET   ;

//-- CIP Communication ---------------------------------------
      AN    DB4331.DBX   15.0;
//      AN "U133SeqD".Seq.PO.B30 // CIP Active (Slave)
      A     #ComCIP;
      JCN   NCIP;
//Conductivity CIP Return
      L     DB4335.DBD  150;
      T     DB4331.DBD  626;

//Temperature CIP Return
      L     DB4335.DBD  146;
      T     DB4331.DBD  594;

//CIP Prerun Pump SP

      CALL FC    45 (
           SFM                      := DB4331.DBD  686,
           Indexes                  := #SFM36);


      L     0.000000e+000;
      A     #SFM36.I01;
      =     DB4335.DBX  171.7;
      JCN   pfc;
      L     DB4331.DBD  654;
pfc:  NOP   0;
      A     #SFM36.I02;
      =     DB4335.DBX  172.0;
      JCN   ppc;
      L     DB4331.DBD  670;
ppc:  NOP   0;
      A     #SFM36.I03;
      =     DB4335.DBX  171.6;
      JCN   pxc;
      L     DB4331.DBD  574;
pxc:  NOP   0;
      T     DB4335.DBD  182;

//CIP Return
      L     DB4331.DBD  558;
      T     DB4335.DBD  186;
      L     DB4335.DBD  138;
      T     DB4331.DBD  562;

//CIP Prerun
      L     DB4331.DBD  542;
      T     DB4335.DBD  190;
      L     DB4335.DBD  142;
      T     DB4331.DBD  546;

// Write Own Data to CIP
      L     DB4335.DBD   10;
      T     DB4335.DBD  154;

      L     DB4335.DBW   14;
      T     DB4335.DBW  158;

      L     DB4335.DBW   16;
      T     DB4335.DBW  160;

      L     DB4335.DBW   18;
      T     DB4335.DBW  162;

      L     DB4335.DBW   20;
      T     DB4335.DBW  164;

      L     DB4335.DBW   22;
      T     DB4335.DBW  166;

      A     DB4335.DBX   24.0;
      =     DB4335.DBX  168.0;

      A     DB4335.DBX   24.1;
      =     DB4335.DBX  168.1;

      A     DB4335.DBX   24.2;
      =     DB4335.DBX  168.2;

      A     DB4335.DBX   24.3;
      =     DB4335.DBX  168.3;

      A     DB4335.DBX   24.4;
      =     DB4335.DBX  168.4;

      A     DB4335.DBX   24.5;
      =     DB4335.DBX  168.5;

      A     DB4335.DBX   24.6;
      =     DB4335.DBX  168.6;

      A     DB4335.DBX   24.7;
      =     DB4335.DBX  168.7;

// Copy Data to CIP
      CALL SFC   20 (
           SRCBLK                   := DB4335.ToCIP,
           RET_VAL                  := #iRetVal,
           DSTBLK                   := DB4335.ToCIP);

NCIP: NOP   0;

//Empty Signal
//A     "U133SpID".SpI.Sig //!!!! Insert correct Empty Signal !!!
      CLR   ;
      =     DB4335.DBX   26.5;

//Full Signal
//A     "U133SpID".SpI.Sig //!!!! Insert correct Full Signal !!!
      CLR   ;
      =     DB4335.DBX   26.2;

//CIP Program Selected
      A     #CIP;
      =     DB4335.DBX   27.1;

// Emergency Stop
      A     #EStopOK; //If needed add or replace with own SpI
      =     DB4335.DBX   27.0; //Emergency Stop OK


NETWORK
TITLE = read from other unit data



END_FUNCTION_BLOCK

FUNCTION_BLOCK FB 4345
TITLE =U134: Planung Transfer D6
FAMILY : BOTEC_F1
NAME : U134Comm
VERSION : 0.1


VAR_TEMP
  iRetVal : INT ;	//return value as integer
  wRetVal : WORD ;	//return value as word
  Run : BOOL ;	//Unit in "RUN" mode
  EStopOK : BOOL ;	//Emergency Stop OK
  CIP : BOOL ;	//CIP Program Selected
  ComCIP : BOOL ;	//Communication with CIP Active
  xTmp : BOOL ;	//Temporary BOOL (free for general use)
  iTmp : INT ;	//Temporary INT (free for general use)
  rTmp : REAL ;	//Temporary REAL (free for general use)
  dTmp : DINT ;	//Temporary DINT (free for general use)
  UnitNo : INT ;	//Unit Number
  EquipmentID : INT ;	//Equipment ID
  Prid : DINT ;	//Process ID
  SFM36 : STRUCT 	// CIP Pump Mode
   I00 : BOOL ;	// Off
   I01 : BOOL ;	// Flow
   I02 : BOOL ;	// Pressure
   I03 : BOOL ;	// Fix Speed
   I04 : BOOL ;
   I05 : BOOL ;
   I06 : BOOL ;
   I07 : BOOL ;
   I08 : BOOL ;
   I09 : BOOL ;
   I10 : BOOL ;
   I11 : BOOL ;
   I12 : BOOL ;
   I13 : BOOL ;
   I14 : BOOL ;
   I15 : BOOL ;
   I16 : BOOL ;
   I17 : BOOL ;
   I18 : BOOL ;
   I19 : BOOL ;
   I20 : BOOL ;
   I21 : BOOL ;
   I22 : BOOL ;
   I23 : BOOL ;
   I24 : BOOL ;
   I25 : BOOL ;
   I26 : BOOL ;
   I27 : BOOL ;
   I28 : BOOL ;
   I29 : BOOL ;
   I30 : BOOL ;
   I31 : BOOL ;
  END_STRUCT ;
END_VAR
BEGIN
NETWORK
TITLE =general

      SET   ;

// unit & equipment number ---------------------------------------------------
      L     DB4340.DBW    0;
      T     #UnitNo;

      L     DB4345.DBW   14;
      L     1000;
      *I    ;
      L     #UnitNo;
      +I    ;
      T     #EquipmentID;

// CIP ----------------------------------------------------------------------
      L     DB4345.DBW   18;
      L     0;
      <I    ;
      =     #CIP;

// Communicating Units-------------------------------------------------------
      L     DB4345.DBD   10;
      L     DB4345.DBD  106;
      ==D   ;
      =     #ComCIP;

// emergency OK -------------------------------------------------------------
      A     DB4345.DBX   75.0; //General Emergency Stop OK
      CLR   ;
      =     #EStopOK;

NETWORK
TITLE =read other unit's data

      SET   ;

// ... General Unit ----------/

      CALL FC   563 (
           ActReq                   := M    101.0,
           PLCNo                    := 3,
           SourceUnitNo             := 99,
           IsTUnit                  := FALSE,
           DstComDRec               := DB4345.GEN,
           RET_VAL                  := #wRetVal);


NETWORK
TITLE =remote start

      SET   ;
// !!! insert correct condition of unit start !!!
      A     DB4341.DBX   15.0;
      A     DB4341.DBX   17.4;
      CLR   ;
      JCN   Strt;
      L     DB4345.DBD   10;
//L        L#-1;                            // Prid negative to start on its own
      T     #Prid;

      CALL FC    48 (
           UnitNo                   := #UnitNo,
           PrId                     := #Prid,
           Run                      := DB4341.DBX   17.4,
           PrIdTransfer             := TRUE,
           Start                    := TRUE,
           RetVal                   := #wRetVal);
Strt: NOP   0;
NETWORK
TITLE =external releases

      SET   ;

NETWORK
TITLE =write own unit data

      SET   ;

//-- CIP Communication ---------------------------------------
      AN    DB4341.DBX   15.0;
//      AN "U134SeqD".Seq.PO.B30 // CIP Active (Slave)
      A     #ComCIP;
      JCN   NCIP;
//Conductivity CIP Return
      L     DB4345.DBD  150;
      T     DB4341.DBD  626;

//Temperature CIP Return
      L     DB4345.DBD  146;
      T     DB4341.DBD  594;

//CIP Prerun Pump SP

      CALL FC    45 (
           SFM                      := DB4341.DBD  686,
           Indexes                  := #SFM36);


      L     0.000000e+000;
      A     #SFM36.I01;
      =     DB4345.DBX  171.7;
      JCN   pfc;
      L     DB4341.DBD  654;
pfc:  NOP   0;
      A     #SFM36.I02;
      =     DB4345.DBX  172.0;
      JCN   ppc;
      L     DB4341.DBD  670;
ppc:  NOP   0;
      A     #SFM36.I03;
      =     DB4345.DBX  171.6;
      JCN   pxc;
      L     DB4341.DBD  574;
pxc:  NOP   0;
      T     DB4345.DBD  182;

//CIP Return
      L     DB4341.DBD  558;
      T     DB4345.DBD  186;
      L     DB4345.DBD  138;
      T     DB4341.DBD  562;

//CIP Prerun
      L     DB4341.DBD  542;
      T     DB4345.DBD  190;
      L     DB4345.DBD  142;
      T     DB4341.DBD  546;

// Write Own Data to CIP
      L     DB4345.DBD   10;
      T     DB4345.DBD  154;

      L     DB4345.DBW   14;
      T     DB4345.DBW  158;

      L     DB4345.DBW   16;
      T     DB4345.DBW  160;

      L     DB4345.DBW   18;
      T     DB4345.DBW  162;

      L     DB4345.DBW   20;
      T     DB4345.DBW  164;

      L     DB4345.DBW   22;
      T     DB4345.DBW  166;

      A     DB4345.DBX   24.0;
      =     DB4345.DBX  168.0;

      A     DB4345.DBX   24.1;
      =     DB4345.DBX  168.1;

      A     DB4345.DBX   24.2;
      =     DB4345.DBX  168.2;

      A     DB4345.DBX   24.3;
      =     DB4345.DBX  168.3;

      A     DB4345.DBX   24.4;
      =     DB4345.DBX  168.4;

      A     DB4345.DBX   24.5;
      =     DB4345.DBX  168.5;

      A     DB4345.DBX   24.6;
      =     DB4345.DBX  168.6;

      A     DB4345.DBX   24.7;
      =     DB4345.DBX  168.7;

// Copy Data to CIP
      CALL SFC   20 (
           SRCBLK                   := DB4345.ToCIP,
           RET_VAL                  := #iRetVal,
           DSTBLK                   := DB4345.ToCIP);

NCIP: NOP   0;

//Empty Signal
//A     "U134SpID".SpI.Sig //!!!! Insert correct Empty Signal !!!
      CLR   ;
      =     DB4345.DBX   26.5;

//Full Signal
//A     "U134SpID".SpI.Sig //!!!! Insert correct Full Signal !!!
      CLR   ;
      =     DB4345.DBX   26.2;

//CIP Program Selected
      A     #CIP;
      =     DB4345.DBX   27.1;

// Emergency Stop
      A     #EStopOK; //If needed add or replace with own SpI
      =     DB4345.DBX   27.0; //Emergency Stop OK


NETWORK
TITLE = read from other unit data



END_FUNCTION_BLOCK

FUNCTION_BLOCK FB 72
TITLE =
AUTHOR : Riedl
FAMILY : BOTEC
NAME : PDAA
VERSION : 2.0

BEGIN
NETWORK
TITLE =

      CALL FC    72 (
           DBConfig                 := DB    72,
           DBData                   := DB    73);

END_FUNCTION_BLOCK

FUNCTION_BLOCK FB 81
TITLE =
AUTHOR : Riedl
FAMILY : BOTEC
NAME : CrCA
VERSION : 2.1


VAR_TEMP
  wTmp : WORD ;
END_VAR
BEGIN
NETWORK
TITLE =transfer data in own Datablock

// Alter DB Doehler Tuch
      CALL FC   564 (
           ActReq                   := M    101.0,
           PLCNo                    := 1,
           SourceAdr                := P#DB834.DBX 0.0 BYTE 64,
           DataLen                  := 64,
           DestAdr                  := P#DB304.DBX0.0 BYTE 64,
           RET_VAL                  := #wTmp);

// Read from PLC04
      CALL FC   564 (
           ActReq                   := M    101.0,
           PLCNo                    := 4,
           SourceAdr                := P#DB302.DBX0.0 BYTE 128,
           DataLen                  := 128,
           DestAdr                  := P#DB302.DBX0.0 BYTE 128,
           RET_VAL                  := #wTmp);

NETWORK
TITLE =Daten An PLC01 (Tuchenhagen Daten)

      CALL FC   999 ;

NETWORK
TITLE =coupling active bits initialize

      AN    M    101.4;
      JC    NCRC;
      R     DB79.DBX   13.4; // initialize active bits (reset)
      R     DB79.DBX   33.4;
      R     DB79.DBX   53.4;
      R     DB79.DBX   73.4;
      R     DB79.DBX   93.4;
      R     DB79.DBX  113.4;
      R     DB79.DBX  133.4;
      R     DB79.DBX  153.4;
      R     DB79.DBX  173.4;
      R     DB79.DBX  193.4;
      R     DB79.DBX  213.4;
      R     DB79.DBX  233.4;
      R     DB79.DBX  253.4;
      R     DB79.DBX  273.4;
      R     DB79.DBX  293.4;
      R     DB79.DBX  313.4;
NCRC: SET   ;
NETWORK
TITLE =read data from remote PLC

      NOP   0;

// From PLC01
//      CALL  "CrC" , "CrCD"
//       RemotePLCNo:=1

// From PLC02
//      CALL  "CrC" , "CrCD"
//       RemotePLCNo:=2

// From PLC03
//     CALL  "CrC" , "CrCD"
//       RemotePLCNo:=3

// From PLC04
      CALL FB    80 , DB    80 (
           RemotePLCNo              := 4);

// From PLC05
//      CALL  "CrC" , "CrCD"
//       RemotePLCNo:=5

// From PLC06
//      CALL  "CrC" , "CrCD"
//       RemotePLCNo:=6

// From PLC07
//      CALL  "CrC" , "CrCD"
//       RemotePLCNo:=7

// From PLC08
//      CALL  "CrC" , "CrCD"
//       RemotePLCNo:=8

// From PLC09
//      CALL  "CrC" , "CrCD"
//       RemotePLCNo:=9

// From PLC10
//      CALL  "CrC" , "CrCD"
//       RemotePLCNo:=10

// From PLC11
//      CALL  "CrC" , "CrCD"
//       RemotePLCNo:=11

// From PLC12
//      CALL  "CrC" , "CrCD"
//       RemotePLCNo:=12

// From PLC13
//      CALL  "CrC" , "CrCD"
//       RemotePLCNo:=13

// From PLC14
//      CALL  "CrC" , "CrCD"
//       RemotePLCNo:=14

// From PLC15
//      CALL  "CrC" , "CrCD"
//       RemotePLCNo:=15

// From PLC16
//      CALL  "CrC" , "CrCD"
//       RemotePLCNo:=16

END_FUNCTION_BLOCK

FUNCTION_BLOCK FB 111
TITLE =C01: Water Tank x
// NW  1 : phase and index evaluation
// NW  2 : phase  1: start position
// NW  3 : phase  4: Filling
// NW  4 : phase  5: Storage
// NW  5 : phase  8: Emptying
// NW  6 : phase 20: Quality Check
// NW  7 : phase 21: Prepare Tank
// NW  8 : phase 23: Connect Tank
// NW  9 : phase 31: CIP Start
// NW 10 : phase 32: CIP Prerun
// NW 11 : phase 33: CIP Return
// NW 12 : phase 34: CIP Rinsing
// NW 13 : phase 35: CIP Emptying
// NW 14 : phase 36: CIP Drain
// NW 15 : phase 40: CIP End
// NW 16 : end of sequence
// NW 17 : unit hold request
//SFM   Use                                 Datatype        UoM
//----+-------------------------------------------------------------------------
// 09 : Process Time                        Duration        min
// 40 : Density                             Value           kg/l
// 42 : Material                            Value
AUTHOR : Woermann
NAME : C01Seq
VERSION : 0.1
CODE_VERSION1


VAR
  U : UDT 111;
END_VAR
VAR_TEMP
  CIP : BOOL ;	//CIP active
  ComCIP : BOOL ;	//Communication With CIP Active
  ComSRC : BOOL ;	//Communication With Well Transfer x
  RRel : BOOL ;	//Run Release
  EStopOK : BOOL ;	//emergency OK
  StepMax : BOOL ;	//StepMax (last) active
  SubStepMax : BOOL ;	//SubStepMax (last) active
  SubStepMaxD : BOOL ;	//SubStepMax (last) done
  ChkOK : BOOL ;	//SubStepMax (last) done
  xTmp : BOOL ;	//Temporary BOOL (free for general use)
  iTmp : INT ;	//Temporary INT (free for general use)
  dTmp : DINT ;	//Temporary DINT (free for general use)
  rTmp : REAL ;	//Temporary REAL (free for general use)
  dUnitNo : DINT ;	//Unit Number
  UnitNo : INT ;	//Unit Number
  EquipmentID : INT ;	//Equipment ID
  S2I : STRUCT 	//SFM to indexes
   SFM26 : STRUCT 	//Cip Step On Condition
    I00 : BOOL ;	//Please Select
    I01 : BOOL ;	//Conductivity High
    I02 : BOOL ;	//Conductivity Low
    I03 : BOOL ;	//Time
    I04 : BOOL ;	//Amount
    I05 : BOOL ;	//Temperature High
    I06 : BOOL ;	//Temperature Low
    I07 : BOOL ;
    I08 : BOOL ;
    I09 : BOOL ;
    I10 : BOOL ;
    I11 : BOOL ;
    I12 : BOOL ;
    I13 : BOOL ;
    I14 : BOOL ;
    I15 : BOOL ;
    I16 : BOOL ;
    I17 : BOOL ;
    I18 : BOOL ;
    I19 : BOOL ;
    I20 : BOOL ;
    I21 : BOOL ;
    I22 : BOOL ;
    I23 : BOOL ;
    I24 : BOOL ;
    I25 : BOOL ;
    I26 : BOOL ;
    I27 : BOOL ;
    I28 : BOOL ;
    I29 : BOOL ;
    I30 : BOOL ;
    I31 : BOOL ;
   END_STRUCT ;
   SFM27 : STRUCT 	//Cip Prerun
    I00 : BOOL ;	//None
    I01 : BOOL ;	//Recovered Water
    I02 : BOOL ;	//Caustic
    I03 : BOOL ;
    I04 : BOOL ;	//Acid
    I05 : BOOL ;
    I06 : BOOL ;
    I07 : BOOL ;
    I08 : BOOL ;
    I09 : BOOL ;
    I10 : BOOL ;
    I11 : BOOL ;
    I12 : BOOL ;	//Fresh Water
    I13 : BOOL ;	//Warm Water
    I14 : BOOL ;
    I15 : BOOL ;
    I16 : BOOL ;
    I17 : BOOL ;
    I18 : BOOL ;
    I19 : BOOL ;
    I20 : BOOL ;
    I21 : BOOL ;
    I22 : BOOL ;
    I23 : BOOL ;
    I24 : BOOL ;
    I25 : BOOL ;
    I26 : BOOL ;
    I27 : BOOL ;
    I28 : BOOL ;
    I29 : BOOL ;
    I30 : BOOL ;
    I31 : BOOL ;
   END_STRUCT ;
   SFM28 : STRUCT 	//Cip Return
    I00 : BOOL ;	//None
    I01 : BOOL ;	//Recovered Water
    I02 : BOOL ;	//Caustic
    I03 : BOOL ;
    I04 : BOOL ;	//Acid
    I05 : BOOL ;
    I06 : BOOL ;
    I07 : BOOL ;
    I08 : BOOL ;
    I09 : BOOL ;
    I10 : BOOL ;
    I11 : BOOL ;
    I12 : BOOL ;	//Fresh Water
    I13 : BOOL ;	//Warm Water
    I14 : BOOL ;
    I15 : BOOL ;	//Drain
    I16 : BOOL ;
    I17 : BOOL ;
    I18 : BOOL ;
    I19 : BOOL ;
    I20 : BOOL ;
    I21 : BOOL ;
    I22 : BOOL ;
    I23 : BOOL ;
    I24 : BOOL ;
    I25 : BOOL ;
    I26 : BOOL ;
    I27 : BOOL ;
    I28 : BOOL ;
    I29 : BOOL ;
    I30 : BOOL ;
    I31 : BOOL ;
   END_STRUCT ;
   SFM37 : STRUCT 	//Cip Pump Mode
    I00 : BOOL ;	//Off
    I01 : BOOL ;	//Flow
    I02 : BOOL ;	//Pressure
    I03 : BOOL ;	//Fix Speed
    I04 : BOOL ;
    I05 : BOOL ;
    I06 : BOOL ;
    I07 : BOOL ;
    I08 : BOOL ;
    I09 : BOOL ;
    I10 : BOOL ;
    I11 : BOOL ;
    I12 : BOOL ;
    I13 : BOOL ;
    I14 : BOOL ;
    I15 : BOOL ;
    I16 : BOOL ;
    I17 : BOOL ;
    I18 : BOOL ;
    I19 : BOOL ;
    I20 : BOOL ;
    I21 : BOOL ;
    I22 : BOOL ;
    I23 : BOOL ;
    I24 : BOOL ;
    I25 : BOOL ;
    I26 : BOOL ;
    I27 : BOOL ;
    I28 : BOOL ;
    I29 : BOOL ;
    I30 : BOOL ;
    I31 : BOOL ;
   END_STRUCT ;
   SFM31 : STRUCT 	//Cip Distribution Circuit No
    I00 : BOOL ;	//Please Select
    I01 : BOOL ;	//Auto Select
    I02 : BOOL ;
    I03 : BOOL ;
    I04 : BOOL ;
    I05 : BOOL ;
    I06 : BOOL ;
    I07 : BOOL ;
    I08 : BOOL ;
    I09 : BOOL ;
    I10 : BOOL ;
    I11 : BOOL ;
    I12 : BOOL ;
    I13 : BOOL ;
    I14 : BOOL ;
    I15 : BOOL ;
    I16 : BOOL ;
    I17 : BOOL ;
    I18 : BOOL ;
    I19 : BOOL ;
    I20 : BOOL ;
    I21 : BOOL ;
    I22 : BOOL ;
    I23 : BOOL ;
    I24 : BOOL ;
    I25 : BOOL ;
    I26 : BOOL ;
    I27 : BOOL ;
    I28 : BOOL ;
    I29 : BOOL ;
    I30 : BOOL ;
    I31 : BOOL ;
   END_STRUCT ;
   SFM39 : STRUCT 	//Q-Status
    I00 : BOOL ;	//Please select
    I01 : BOOL ;	//released
    I02 : BOOL ;
    I03 : BOOL ;
    I04 : BOOL ;
    I05 : BOOL ;
    I06 : BOOL ;	//Ignore
    I07 : BOOL ;
    I08 : BOOL ;
    I09 : BOOL ;	//locked
    I10 : BOOL ;
    I11 : BOOL ;
    I12 : BOOL ;
    I13 : BOOL ;
    I14 : BOOL ;
    I15 : BOOL ;
    I16 : BOOL ;
    I17 : BOOL ;
    I18 : BOOL ;
    I19 : BOOL ;
    I20 : BOOL ;
    I21 : BOOL ;
    I22 : BOOL ;
    I23 : BOOL ;
    I24 : BOOL ;
    I25 : BOOL ;
    I26 : BOOL ;
    I27 : BOOL ;
    I28 : BOOL ;
    I29 : BOOL ;
    I30 : BOOL ;
    I31 : BOOL ;
   END_STRUCT ;
  END_STRUCT ;
  ComDST : BOOL ;	//Communication Water Transfer to Packaging Plant
  ComCIPDist : BOOL ;	//Communication with CIP Distribution
  ReqInlet : BOOL ;	//Request Inlet
  RelOutlet : BOOL ;	//Release Outlet
  Empty : BOOL ;	//Tank Empty
  reqAnlage : BOOL ;	//Destination Requests Filling
  ComU043 : BOOL ;
  ComU045 : BOOL ;
  ComU047 : BOOL ;
  ComU048 : BOOL ;
  ComU049 : BOOL ;
  ComU050 : BOOL ;
  ComU051 : BOOL ;
  ComU052 : BOOL ;
  ComU054 : BOOL ;
  ComU055 : BOOL ;
  ComU056 : BOOL ;
  ComU057 : BOOL ;
  ComU058 : BOOL ;
  ComLine : INT ;	//Check Line Communikation and send to all lines
END_VAR
BEGIN
NETWORK
TITLE = Phase and Index Evaluation


      CLR   ;
      =     #RRel;
      =     #ReqInlet;
      =     #RelOutlet;
      L     0;
      T     #ComLine;

// ---------------------------------------------------------------------------
// write max used SFM's (last SFM number + 1)
      L     60;
      T     #U.SFMQuant;

// ---------------------------------------------------------------------------
// unit & equipment number
      L     MB   112;
      T     #UnitNo;

      L     DB115.DBW   14;
      L     1000;
      *I    ;
      L     #UnitNo;
      +I    ;
      T     #EquipmentID;

// ---------------------------------------------------------------------------
// CIP active
      L     MW   114;
      L     0;
      <I    ;
      =     #CIP;

// ---------------------------------------------------------------------------
// communicating units
      L     MD   124;
      L     DB115.DBD  106;
      ==D   ;
      =     #ComCIP;

      L     MD   124;
      L     DB1945.DBD   10; // CIP Dist 1
      ==D   ;
      =     #ComCIPDist;

      A(    ;
      L     DB115.DBD  226;
      RND   ;
      L     #EquipmentID;
      ==D   ;
      )     ;
      A(    ;
      L     #U.Seq.SFM[42].Sp; // Material
      L     DB115.DBD  222;
      ==R   ;
      )     ;
      =     #ComSRC;




      CLR   ;
      A(    ; // Material Check
      L     #U.Seq.SFM[42].Sp; // Material
      L     DB1435.DBD   30;
      ==R   ;
      )     ;
      A(    ;
      L     DB1435.DBD   34;
      RND   ;
      L     #EquipmentID;
      ==R   ;
      )     ;
      =     #ComU043;

      A(    ; // Material Check
      L     #U.Seq.SFM[42].Sp; // Material
      L     DB1455.DBD   30;
      ==R   ;
      )     ;
      A(    ;
      L     DB1455.DBD   34;
      RND   ;
      L     #EquipmentID;
      ==R   ;
      )     ;
      =     #ComU045;

      A(    ; // Material Check
      L     #U.Seq.SFM[42].Sp; // Material
      L     DB1475.DBD   30;
      ==R   ;
      )     ;
      A(    ;
      L     DB1475.DBD   34;
      RND   ;
      L     #EquipmentID;
      ==R   ;
      )     ;
      =     #ComU047;

      A(    ; // Material Check
      L     #U.Seq.SFM[42].Sp; // Material
      L     DB1485.DBD   30;
      ==R   ;
      )     ;
      A(    ;
      L     DB1485.DBD   34;
      RND   ;
      L     #EquipmentID;
      ==R   ;
      )     ;
      =     #ComU048;

      A(    ; // Material Check
      L     #U.Seq.SFM[42].Sp; // Material
      L     DB1495.DBD   30;
      ==R   ;
      )     ;
      A(    ;
      L     DB1495.DBD   34;
      RND   ;
      L     #EquipmentID;
      ==R   ;
      )     ;
      =     #ComU049;

      A(    ; // Material Check
      L     #U.Seq.SFM[42].Sp; // Material
      L     DB1505.DBD   30;
      ==R   ;
      )     ;
      A(    ;
      L     DB1505.DBD   34;
      RND   ;
      L     #EquipmentID;
      ==R   ;
      )     ;
      =     #ComU050;

      A(    ; // Material Check
      L     #U.Seq.SFM[42].Sp; // Material
      L     DB1515.DBD   30;
      ==R   ;
      )     ;
      A(    ;
      L     DB1515.DBD   34;
      RND   ;
      L     #EquipmentID;
      ==R   ;
      )     ;
      =     #ComU051;

      A(    ; // Material Check
      L     #U.Seq.SFM[42].Sp; // Material
      L     DB1525.DBD   30;
      ==R   ;
      )     ;
      A(    ;
      L     DB1525.DBD   34;
      RND   ;
      L     #EquipmentID;
      ==R   ;
      )     ;
      =     #ComU052;

      A(    ; // Material Check
      L     #U.Seq.SFM[42].Sp; // Material
      L     DB1545.DBD   30;
      ==R   ;
      )     ;
      A(    ;
      L     DB1545.DBD   34;
      RND   ;
      L     #EquipmentID;
      ==R   ;
      )     ;
      =     #ComU054;

      A(    ; // Material Check
      L     #U.Seq.SFM[42].Sp; // Material
      L     DB1555.DBD   30;
      ==R   ;
      )     ;
      A(    ;
      L     DB1555.DBD   34;
      RND   ;
      L     #EquipmentID;
      ==R   ;
      )     ;
      =     #ComU055;

      A(    ; // Material Check
      L     #U.Seq.SFM[42].Sp; // Material
      L     DB1565.DBD   30;
      ==R   ;
      )     ;
      A(    ;
      L     DB1565.DBD   34;
      RND   ;
      L     #EquipmentID;
      ==R   ;
      )     ;
      =     #ComU056;

      A(    ; // Material Check
      L     #U.Seq.SFM[42].Sp; // Material
      L     DB1575.DBD   30;
      ==R   ;
      )     ;
      A(    ;
      L     DB1575.DBD   34;
      RND   ;
      L     #EquipmentID;
      ==R   ;
      )     ;
      =     #ComU057;

      A(    ; // Material Check
      L     #U.Seq.SFM[42].Sp; // Material
      L     DB1585.DBD   30;
      ==R   ;
      )     ;
      A(    ;
      L     DB1585.DBD   34;
      RND   ;
      L     #EquipmentID;
      ==R   ;
      )     ;
      =     #ComU058;



      CLR   ;
      =     #ComDST;

// Release Emptying / Filling of Tank ----------------------------------------
      A     DB211.DBX   78.7;
      =     M    130.3; // Delay Empty

      A     M    152.1; // Filling Release
      S     #U.Seq.User.Bit5;
      AN    DB211.DBX  138.7; // Full False
      R     #U.Seq.User.Bit5;

      A     M    152.2; // Emptying Release
      ON    DB115.DBX  218.3;
      S     #U.Seq.User.Bit6;
      A     M    150.3; // Empty True
      R     #U.Seq.User.Bit6;

// ---------------------------------------------------------------------------
// process timer start
      SET   ;
      =     M    131.0;

// ---------------------------------------------------------------------------
// emergency OK
      A     DB115.DBX   27.0;
      =     #EStopOK;

// define last (Sub)Step active
      L     #U.Seq.StepMax;
      L     MW   104;
      ==I   ;
      =     #StepMax;

      L     #U.Seq.SubStepMax;
      L     MW   118;
      ==I   ;
      =     #SubStepMax;

      A     #SubStepMax;
      A     #U.Seq.SPD;
      AN    M    103.2;
      =     #SubStepMaxD;

// ---------------------------------------------------------------------------
// phase evaluation
      L     MW   108;
      JL    X0;
      JU    X0; // phase  0:
      JU    X1; // phase  1: start position
      JU    X0; // phase  2:
      JU    X0; // phase  3:
      JU    X4; // phase  4: Filling
      JU    X5; // phase  5: Storage
      JU    X0; // phase  6:
      JU    X0; // phase  7:
      JU    X8; // phase  8: Emptying
      JU    X0; // phase  9:
      JU    X0; // phase 10:
      JU    X0; // phase 11:
      JU    X0; // phase 12:
      JU    X0; // phase 13:
      JU    X0; // phase 14:
      JU    X0; // phase 15:
      JU    X0; // phase 16:
      JU    X0; // phase 17:
      JU    X0; // phase 18:
      JU    X0; // phase 19:
      JU    X20; // phase 20: Quality Check
      JU    X21; // phase 21: Prepare Tank
      JU    X0; // phase 22:
      JU    X23; // phase 23: Connect Tank
      JU    X0; // phase 24:
      JU    X0; // phase 25:
      JU    X0; // phase 26:
      JU    X0; // phase 27:
      JU    X0; // phase 28:
      JU    X0; // phase 29:
      JU    X0; // phase 30:
      JU    X31; // phase 31: CIP Start
      JU    X32; // phase 32: CIP Prerun
      JU    X33; // phase 33: CIP Return
      JU    X34; // phase 34: CIP Rinsing
      JU    X35; // phase 35: CIP Emptying
      JU    X36; // phase 36: CIP Drain
      JU    X0; // phase 37:
      JU    X0; // phase 38:
      JU    X0; // phase 39:
      JU    X40; // phase 40: CIP End
X0:   SET   ;
      S     M    108.7; // Error unknown phase
      JU    COMM;
NETWORK
TITLE =phase 1: startposition

X1:   SET   ;

// ---------------------------------------------------------------------------
// general functions
// ---------------------------------------------------------------------------
// reset signals
      A     M    102.2;
      R     #U.Seq.Switch.Sw1;
      R     #U.Seq.Switch.Sw2;

      AN    M    102.0;
      =     M    161.0; // Reset Process Timer

      CALL FC   709 (// Reset "Simulation" And "Ignore"
           UnitNo                   := #UnitNo,// Of All Control Modules
           Enable                   := M    102.2);// At First Cycle of Startposition (Idle)

// ---------------------------------------------------------------------------
// start check --------------------------------------------------------------
      A     #CIP;
      JC    M010;

      CALL FC   110 (
           ChkType                  := 1,// production
           ChkOK                    := M    122.0);
      JU    COMM;

M010: CALL FC   110 (
           ChkType                  := 2,// CIP
           ChkOK                    := M    122.0);
      JU    COMM;
NETWORK
TITLE =phase 4: Filling
//SFM   Use                                 Datatype        UoM
//----+-------------------------------------------------------------------------
// 00 : Watch Dog Time                      Duration        min
// 17 : Level                               Value           l
X4:   SET   ;
// ---------------------------------------------------------------------------
// General CM evaluation
      CALL FC   110 (
           ChkType                  := 3,
           ChkOK                    := #ChkOK);

      AN    #ChkOK;
      S     M    120.3;

// ---------------------------------------------------------------------------
// general functions
      AN    M    121.2;
      A     M    102.3;
      =     #RRel;

      A     M    102.3;
      =     DB115.DBX   26.0;

// ---------------------------------------------------------------------------
// messages
// ---------------------------------------------------------------------------
// timer & counter
      A     M    102.0;

// ---------------------------------------------------------------------------
// pause timer
// ---------------------------------------------------------------------------
// communication

// ---------------------------------------------------------------------------
// control modules

// ---------------------------------------------------------------------------
// transition condition
      A     #U.Seq.User.Bit6; // EMPTY_REL
      AN    M    102.2;
      =     M    102.1;


// ---------------------------------------------------------------------------
// ---------------------------------------------------------------------------
// subphase repeat function
      A     #SubStepMax;
      JCN   Y4;
      L     1;
      T     MW   116;
Y4:   SET   ;

// subphase evaluation
      L     MW   110;
      JL    A400;
      JU    COMM; // subphase  0:
      JU    A401; // subphase  1: Waiting
      JU    A402; // subphase  2: Active
// ---------------------------------------------------------------------------
A400: SET   ;
      S     M    110.7; // Error unknown subphase
      JU    COMM;

// subphase 1: Waiting
A401: SET   ;
// -------------------------------------------------
// subphase timer & counter
      A     M    103.0;

// -------------------------------------------------
// subphase actuator


// -------------------------------------------------
// subphase transition
      A     DB115.DBX  218.4;
      A     #ComSRC;
      AN    M    103.2;
      =     M    103.1;
      JU    COMM;

// subphase 2: Active
A402: SET   ;
      A     #U.Seq.User.Bit2;
      A     M    103.3;
      =     DB115.DBX   26.1;
// -------------------------------------------------
// subphase timer & counter
      A     M    103.0;

// -------------------------------------------------
// subphase actuator
      A     M    103.3;
      =     #ReqInlet;
// -------------------------------------------------
// subphase transition
      AN    DB115.DBX  218.4;
      ON    #ComSRC;
      =     M    103.1;
      JU    COMM;
NETWORK
TITLE =phase 5: Production
//SFM   Use                                 Datatype        UoM
//----+-------------------------------------------------------------------------
// 00 : Watch Dog Time                      Duration        min
// 05 : Substep Time                        Duration        s
// 17 : Level                               Value           l
X5:   SET   ;
// ---------------------------------------------------------------------------
// General CM evaluation
      CALL FC   110 (
           ChkType                  := 3,
           ChkOK                    := #ChkOK);

      AN    #ChkOK;
      S     M    120.3;

// ---------------------------------------------------------------------------
// general functions
      AN    M    121.2;
      A     M    102.3;
      =     #RRel;

      A     M    102.3;
      =     DB115.DBX   26.3;

// ---------------------------------------------------------------------------
// messages
// ---------------------------------------------------------------------------
// timer & counter
      A     M    102.0;

// ---------------------------------------------------------------------------
// pause timer
      ON    M    102.3;
      O     M    150.4;
      S     M    140.4; // Substep Time

// ---------------------------------------------------------------------------
// communication
      A     DB1435.DBX   26.1;
      A     #ComU043;
      O     ;
      A     DB1455.DBX   26.1;
      A     #ComU045;
      O     ;
      A     DB1475.DBX   26.1;
      A     #ComU047;
      O     ;
      A     DB1485.DBX   26.1;
      A     #ComU048;
      O     ;
      A     DB1495.DBX   26.1;
      A     #ComU049;
      O     ;
      A     DB1505.DBX   26.1;
      A     #ComU050;
      O     ;
      A     DB1515.DBX   26.1;
      A     #ComU051;
      O     ;
      A     DB1525.DBX   26.1;
      A     #ComU052;
      O     ;
      A     DB1545.DBX   26.1;
      A     #ComU054;
      O     ;
      A     DB1555.DBX   26.1;
      A     #ComU055;
      O     ;
      A     DB1565.DBX   26.1;
      A     #ComU056;
      O     ;
      A     DB1575.DBX   26.1;
      A     #ComU057;
      O     ;
      A     DB1585.DBX   26.1;
      A     #ComU058;
      =     #reqAnlage;



// ---------------------------------------------------------------------------
// control modules
      A     M    102.3;

// ---------------------------------------------------------------------------
// transition condition
      AN    #U.Seq.User.Bit5; // FILL_REL
      ON    #U.Seq.User.Bit6; // EMPTY_REL
      AN    M    102.2;
      =     M    102.1;

      AN    #U.Seq.User.Bit6; // EMPTY_REL
      JCN   N401; // GoTo Filling
      L     MW   104;
      L     1;
      -I    ;
      T     MW   106;
N401: SET   ;

// ---------------------------------------------------------------------------
// ---------------------------------------------------------------------------
// subphase repeat function
      A     #SubStepMax;
      JCN   Y5;
      L     1;
      T     MW   116;
Y5:   SET   ;

// subphase evaluation
      L     MW   110;
      JL    A500;
      JU    COMM; // subphase  0:
      JU    A501; // subphase  1: Waiting
      JU    A502; // subphase  2: Active
// ---------------------------------------------------------------------------
A500: SET   ;
      S     M    110.7; // Error unknown subphase
      JU    COMM;

// subphase 1: Waiting
A501: SET   ;
      A     M    103.3;
      =     DB115.DBX   26.0;
      R     DB115.DBX   26.4;
// -------------------------------------------------
// subphase timer & counter
      A     M    103.0;

// -------------------------------------------------
// subphase actuator
      A     M    103.3;

// -------------------------------------------------
// subphase transition
      A     #reqAnlage;
      O     DB115.DBX  218.4;
      =     M    103.1;
      JU    COMM;

// subphase 2: Active
A502: SET   ;
// Communication Filling
      A     #U.Seq.User.Bit2;
      A     M    103.3;
      =     DB115.DBX   26.1;

      AN    DB115.DBX  218.4;
      A     M    103.3;
      =     DB115.DBX   26.0;

// Communication Emptying

      A     M    103.3;
      =     DB115.DBX   26.3;

// -------------------------------------------------
// subphase timer & counter
      A     M    103.0;

// -------------------------------------------------
// subphase actuator


// Emptying -------------
      CLR   ;
      =     DB115.DBX   26.4;
//KEG
      A     DB1435.DBX   26.1;
      A     #ComU043;
      A     M    103.3;
      =     DB210.DBX  268.0;

      A     DB210.DBX  268.0;
      A     DB210.DBX  262.6;
      S     DB115.DBX   26.4;
      JCN   A3rm;
      L     #ComLine;
      L     1;
      OW    ;
      T     #ComLine;
A3rm: NOP   0;
//A5
      A     DB1455.DBX   26.1;
      A     #ComU045;
      A     M    103.3;
      =     DB210.DBX  828.0;

      A     DB210.DBX  828.0;
      A     DB210.DBX  822.6;
      S     DB115.DBX   26.4;
      JCN   A5rm;
      L     #ComLine;
      L     2;
      OW    ;
      T     #ComLine;
A5rm: NOP   0;

//A7
      A     DB1475.DBX   26.1;
      A     #ComU047;
      A     M    103.3;
      =     DB210.DBX  668.0;

      A     DB210.DBX  668.0;
      A     DB210.DBX  662.6;
      S     DB115.DBX   26.4;
      JCN   A7rm;
      L     #ComLine;
      L     4;
      OW    ;
      T     #ComLine;
A7rm: NOP   0;

//A9
      A     DB1495.DBX   26.1;
      A     #ComU049;
      A     M    103.3;
      =     DB210.DBX  508.0;

      A     DB210.DBX  508.0;
      A     DB210.DBX  502.6;
      S     DB115.DBX   26.4;
      JCN   A9rm;
      L     #ComLine;
      L     8;
      OW    ;
      T     #ComLine;
A9rm: NOP   0;

//A10
      A     DB1505.DBX   26.1;
      A     #ComU050;
      A     M    103.3;
      =     DB210.DBX  428.0;

      A     DB210.DBX  428.0;
      A     DB210.DBX  422.6;
      S     DB115.DBX   26.4;
      JCN   AArm;
      L     #ComLine;
      L     16;
      OW    ;
      T     #ComLine;
AArm: NOP   0;

//A11
      A     DB1515.DBX   26.1;
      A     #ComU051;
      A     M    103.3;
      =     DB210.DBX  908.0;

      A     DB210.DBX  908.0;
      A     DB210.DBX  902.6;
      S     DB115.DBX   26.4;
      JCN   ABrm;
      L     #ComLine;
      L     32;
      OW    ;
      T     #ComLine;
ABrm: NOP   0;

//A12
      A     DB1525.DBX   26.1;
      A     #ComU052;
      A     M    103.3;
      =     DB210.DBX  588.0;

      A     DB210.DBX  588.0;
      A     DB210.DBX  582.6;
      S     DB115.DBX   26.4;
      JCN   ACrm;
      L     #ComLine;
      L     64;
      OW    ;
      T     #ComLine;
ACrm: NOP   0;

//A14
      A     DB1545.DBX   26.1;
      A     #ComU054;
      A     M    103.3;
      =     DB210.DBX  988.0;

